Yaskawa INFORM job: OK_R2_O8A-O21A(90,0)OKKR.JBI

/JOB
//NAME OK_R2_O8A-O21A(90,0)OKKR
///FOLDERNAME X4
//POS
///NPOS 715,715,715,30,0,0
///TOOL 0
///POSTYPE PULSE
///PULSE
C00000=-132511,-103668,-126871,1472,79341,-68717
C00001=-132511,-105453,-125920,1479,77839,-68735
C00002=-149942,-121925,-119361,-5630,57848,-69572
C00003=-131289,-120708,-115141,-16553,58451,-62255
C00004=-130492,-107448,-108919,-16502,61476,-62404
C00005=-130492,-107531,-107691,-16624,60708,-62286
C00006=-130492,-107522,-107880,-16606,60824,-62304
C00007=-130122,-101219,-105586,-16530,62651,-62436
C00008=-130467,-107013,-108826,-16492,61638,-62417
C00009=-119884,-107962,-112031,-5369,66225,-56914
C00010=-116096,-92200,-106106,-6995,70935,-55838
C00011=-116096,-92633,-105187,-7026,70153,-55791
C00012=-116096,-92564,-105343,-7022,70283,-55799
C00013=-116785,-88340,-103625,-6657,71334,-56095
C00014=-116573,-89121,-105150,-6736,71883,-56054
C00015=-146016,-80865,-95606,32019,76533,-60687
C00016=-144125,-79506,-95002,31288,76137,-60071
C00017=-145805,-80719,-95541,31939,76487,-60619
C00018=-143803,-87593,-101078,23589,73333,-61663
C00019=-130467,-106338,-112373,-16140,64070,-62776
C00020=-173804,-84257,-100337,8034,65857,-78258
C00021=-173658,-84030,-99866,7982,65672,-78220
C00022=-173658,-84451,-98929,8028,64885,-78273
C00023=-173658,-84370,-99117,8019,65041,-78263
C00024=-172100,-80256,-97322,7106,65901,-77657
C00025=-174189,-84275,-102553,8181,67232,-78295
C00026=-146680,-106555,-114552,-7207,63010,-68642
C00027=-194694,-79170,-110255,-25784,98520,48468
C00028=-198558,-80793,-107909,-24687,95396,47836
C00029=-200090,-81195,-106872,-24266,94212,47563
C00030=-202263,-84154,-108139,-23691,92956,47080
C00031=-202263,-85492,-106716,-23644,91519,47366
C00032=-203864,-86202,-108997,-23266,92055,46716
C00033=-200090,-81195,-106872,-24266,94212,47563
C00034=-174358,-91389,-89628,-58384,85447,80654
C00035=-175228,-93280,-90391,-58296,84646,80691
C00036=-174358,-91389,-89628,-58384,85447,80654
C00037=-168427,-86826,-93699,-59246,91643,79819
C00038=-162839,-83719,-106729,-43881,81993,66911
C00039=-147123,-91237,-114479,-20257,52031,49855
C00040=-112908,-124838,-130477,-22240,82773,36203
C00041=-117493,-120147,-121828,-21064,78888,35282
C00042=-131517,-88028,-114974,-8271,96172,30135
C00043=-131517,-89283,-114090,-8245,94996,30214
C00044=-131517,-88930,-114352,-8253,95335,30191
C00045=-131178,-82908,-111873,-8367,96921,30191
C00046=-131517,-87249,-115462,-8285,96867,30089
C00047=-132831,-90163,-114266,-11578,93705,29175
C00048=-134095,-89636,-114054,-11263,93680,28777
C00049=-131312,-89742,-115220,-11972,94693,29560
C00050=-110699,-95947,-121920,-22827,92218,35184
C00051=-159423,-136044,-122705,-19473,51748,49954
C00052=-156084,-144100,-135379,-20578,56007,50549
C00053=-159635,-139405,-132559,-18260,112136,84879
C00054=-178843,-153016,-133090,-20490,101295,79475
C00055=-178843,-153131,-133279,-20494,101347,79466
C00056=-178843,-151887,-131264,-20445,100783,79562
C00057=-178843,-153131,-133279,-20494,101347,79466
C00058=-178681,-162456,-135669,-20227,98263,80057
C00059=-165549,-147119,-131679,-18745,106518,83551
C00060=-164263,-165353,-136391,-17937,100651,41944
C00061=-168242,-162829,-132237,-18538,98565,40818
C00062=-170474,-158220,-131092,-19006,99630,39839
C00063=-168242,-162829,-132237,-18538,98565,40818
C00064=-163940,-146805,-133599,-18623,108164,40895
C00065=-162398,-133850,-130940,-19068,113277,40626
C00066=-162571,-113567,-127717,-17378,114163,86924
C00067=-160654,-117481,-127396,-16916,112431,87902
C00068=-160654,-117651,-127195,-16888,112229,87933
C00069=-160654,-118532,-125995,-16733,111086,88103
C00070=-160654,-118346,-126273,-16766,111343,88065
C00071=-161650,-123459,-127890,-16641,109583,87959
C00072=-158594,-113131,-127392,-17075,114977,88272
C00073=-174543,-100010,-122844,-18621,115499,82286
C00074=-174543,-100010,-122844,-18621,115499,82286
C00075=-174543,-100010,-122844,-18621,115499,22315
C00076=-138816,-129701,-130055,-13678,112254,36070
C00077=-137500,-131474,-125884,-13183,109137,36932
C00078=-137500,-131471,-125777,-13177,109074,36939
C00079=-139149,-130411,-125460,-13458,109147,36324
C00080=-137500,-131471,-125777,-13177,109074,36939
C00081=-137500,-129047,-134180,-13875,115320,36192
C00082=-137500,-130207,-132407,-13667,113680,36396
C00083=-137899,-129904,-132317,-13740,113712,36243
C00084=-137899,-129904,-132317,-13740,113712,68510
C00085=-153549,-123160,-126704,-15778,110958,63049
C00086=-153549,-123239,-126516,-15760,110807,63070
C00087=-153549,-123761,-124983,-15622,109641,63231
C00088=-153549,-123239,-126516,-15760,110807,63070
C00089=-162223,-110280,-122283,-17095,113025,59536
C00090=-162223,-111585,-120346,-16843,111240,59807
C00091=-163386,-116637,-122034,-16744,109515,59637
C00092=-162108,-110157,-121578,-17034,112692,59632
C00093=-164629,-100924,-122013,-18009,116976,58006
C00094=-164629,-100924,-122013,-18009,116976,86315
C00095=-166469,-102657,-116169,-17620,113433,86211
C00096=-165427,-104649,-116407,-17406,112807,86697
C00097=-165427,-101226,-120322,-18070,116786,86050
C00098=-165427,-100996,-120510,-18111,117009,86012
C00099=-148525,-143011,-136643,3983,84771,-6637
C00100=-128066,-147732,-136598,30045,86114,-11272
C00101=-107762,-175532,-134890,18909,55578,3499
C00102=-107762,-174389,-134000,18900,55616,3506
C00103=-107762,-171707,-131824,18892,55653,3513
C00104=-107762,-174389,-134000,18900,55616,3506
C00105=-110240,-168768,-132692,19371,58166,2939
C00106=-107762,-174389,-134000,18900,55616,3506
C00107=-136558,-139033,-124155,30771,85335,-13620
C00108=-136645,-139245,-122439,30816,84359,-13917
C00109=-135016,-140023,-122655,30663,83532,-13499
C00110=-136645,-139245,-122439,30816,84359,-13917
C00111=-136645,-142239,-130726,30739,87441,-13088
C00112=-136645,-142239,-130726,30739,87441,-13088
C00113=-136231,-126717,-125654,30746,91494,-11840
C00114=-98133,-136848,-119853,-8087,80711,-399
C00115=-120576,-107226,-130969,4806,98429,26759
C00116=-134040,-103912,-127141,12417,95216,42526
C00117=-135128,-102736,-122709,12628,93295,41985
C00118=-135270,-98410,-119352,12667,93467,41957
C00119=-135270,-99211,-118697,12651,92671,41876
C00120=-135270,-98984,-118890,12655,92901,41899
C00121=-134962,-94751,-117294,12605,94023,42111
C00122=-135502,-100967,-121058,12716,93242,41857
C00123=-134459,-102900,-122675,12466,93098,42180
C00124=-132900,-95838,-124142,12211,97313,43092
C00125=-133104,-101231,-126476,12555,90730,41824
C00126=-142488,-103018,-116603,-18920,70477,-33231
C00127=-149408,-93922,-109008,-15541,69095,-35470
C00128=-149408,-94512,-107956,-15635,68178,-35347
C00129=-149408,-94372,-108222,-15611,68405,-35378
C00130=-148690,-90146,-106536,-15855,69631,-35290
C00131=-149408,-93897,-109054,-15536,69135,-35476
C00132=-123067,-90692,-110186,-27168,77789,-27787
C00133=-102416,-91941,-110630,-34518,86135,-22666
C00134=-101917,-92285,-106963,-34730,79171,-22421
C00135=-101917,-92861,-105821,-34832,78340,-22159
C00136=-102166,-91294,-105409,-34682,78702,-22372
C00137=-102552,-87773,-103968,-34461,79319,-22719
C00138=-102166,-90677,-106542,-34586,79544,-22637
C00139=-88745,-139673,-123014,-32701,61923,-22452
C00140=-91020,-118461,-119227,-25559,70043,-27274
C00141=-91020,-118666,-117531,-25735,69003,-27036
C00142=-91020,-118652,-117696,-25718,69101,-27059
C00143=-92656,-112693,-115717,-24791,70291,-27955
C00144=-91020,-118652,-117696,-25718,69101,-27059
C00145=-83494,-110253,-114881,-28187,73796,-25285
C00146=-83494,-110339,-114551,-28219,73576,-25230
C00147=-84308,-111339,-114895,-27963,73042,-25409
C00148=-86719,-114160,-115853,-27192,71497,-25959
C00149=-85916,-112867,-117155,-27291,73063,-26031
C00150=-123117,-127863,-126220,-28315,69551,-25784
C00151=-125315,-122167,-126738,-14196,74486,-31169
C00152=-125647,-109964,-126758,6698,85320,-36650
C00153=-127309,-126191,-121158,24496,77378,-41430
C00154=-122509,-120998,-116871,23174,76039,-39921
C00155=-117160,-104372,-112630,18566,82677,-37125
C00156=-117160,-104907,-110988,18612,81456,-37312
C00157=-117160,-104733,-111581,18595,81887,-37246
C00158=-112842,-111563,-113988,14481,77147,-33000
C00159=-113063,-106504,-112219,14479,78650,-32898
C00160=-112842,-111563,-113988,14481,77147,-33000
C00161=-122612,-110522,-114147,22924,79491,-39282
C00162=-127138,-114707,-118233,24171,81082,-40600
C00163=-112168,-135147,-125869,19703,71474,-13622
C00164=-107112,-124941,-122811,17686,73526,-11445
C00165=-98892,-86649,-110918,2998,94873,14107
C00166=-112057,-63273,-99647,16927,107898,-6848
C00167=-111820,-63961,-99109,16821,107199,-6872
C00168=-111820,-65039,-98309,16715,106195,-7017
C00169=-111820,-64914,-98405,16727,106313,-7000
C00170=-110559,-64565,-98232,16557,106153,-6607
C00171=-111820,-64402,-98791,16776,106793,-6930
C00172=-102401,-90236,-113117,-129,94163,18304
C00173=-122722,-94557,-112635,4536,92169,11873
C00174=-122722,-95060,-112012,4533,91529,11850
C00175=-122722,-94938,-112169,4534,91688,11856
C00176=-124421,-94788,-112110,4914,91823,11321
C00177=-122722,-94458,-112752,4538,92292,11877
C00178=-121995,-82445,-116286,4470,100580,12401
C00179=-106227,-105095,-124470,-409,77251,17488
C00180=-147196,-120547,-129970,-14917,75808,13222
C00181=-161004,-130220,-121828,-20444,67155,12825
C00182=-163784,-117907,-115753,-19016,68936,11464
C00183=-171500,-102190,-112609,-10247,77482,8342
C00184=-172766,-99537,-110960,-8908,78464,7982
C00185=-164799,-113448,-113379,-18515,69495,10996
C00186=-160173,-111708,-112729,-20272,71037,12446
C00187=-159937,-107532,-111273,-20230,72269,12319
C00188=-160173,-111708,-112729,-20272,71037,12446
C00189=-157530,-113449,-113320,-21331,71196,13397
C00190=-157502,-114878,-111335,-21583,69377,13748
C00191=-159463,-112600,-110567,-20755,69532,12980
C00192=-157502,-114878,-111335,-21583,69377,13748
C00193=-157530,-113449,-113320,-21331,71196,13397
C00194=-164799,-113448,-113379,-18515,69495,10996
C00195=-163784,-117907,-115753,-19016,68936,11464
C00196=-161004,-130220,-121828,-20444,67155,12825
C00197=-158635,-143974,-124952,-47178,64629,-48132
C00198=-161510,-136095,-119169,-46184,63472,-49060
C00199=-162608,-132555,-115350,-46042,62530,-49158
C00200=-162346,-131008,-113540,-46239,62439,-48970
C00201=-162608,-133192,-116899,-45817,62973,-49385
C00202=-136560,-74570,-80638,-73986,100743,-31924
C00203=-136560,-74368,-74379,-73183,99581,-30233
C00204=-138115,-75223,-74700,-73053,98436,-30293
C00205=-135508,-73752,-74143,-73275,100358,-30196
C00206=-149616,-145660,-96573,-81184,49972,-24507
C00207=-150329,-142641,-96001,-80244,49710,-25268
C00208=-148962,-149729,-97186,-82532,50127,-23453
C00209=-146770,-153464,-99018,-82858,51507,-22849
C00210=-140616,-162996,-103531,-83341,55379,-21287
C00211=-129649,-178931,-115518,-81569,62637,-20208
C00212=-149811,-117254,-127694,-14309,93218,-9052
C00213=-138773,-86779,-112433,-16512,101214,-6420
C00214=-139010,-84837,-109587,-16423,100448,-6393
C00215=-139010,-86284,-108173,-16326,98898,-6181
C00216=-139046,-85929,-108499,-16342,99259,-6242
C00217=-139851,-81484,-106752,-16280,100273,-6644
C00218=-139210,-85073,-109125,-16364,100022,-6400
C00219=-160229,-93267,-112119,-12359,94277,-12585
C00220=-159749,-92653,-111811,-12461,94470,-12448
C00221=-159749,-93339,-110977,-12438,93625,-12360
C00222=-159895,-92298,-111808,-12436,94626,-12511
C00223=-160151,-89339,-110624,-12406,95366,-12669
C00224=-159895,-92298,-111808,-12436,94626,-12511
C00225=-154010,-101242,-121994,-13665,97135,-10872
C00226=-154083,-100267,-121778,-13665,97483,-10934
C00227=-147006,-81102,-116195,-13282,100818,40144
C00228=-151269,-63896,-105225,-12354,102282,38687
C00229=-152138,-63686,-103764,-12097,101397,38514
C00230=-152138,-64898,-103136,-12048,100410,38612
C00231=-152138,-64707,-103240,-12056,100569,38597
C00232=-153752,-65312,-103536,-11647,100239,38140
C00233=-152274,-63472,-103683,-12067,101440,38470
C00234=-162010,-107602,-126737,-9369,91949,36281
C00235=-162010,-107602,-126737,-9369,91949,36281
C00236=-210314,-79584,-107375,35746,108623,-54127
C00237=-185587,-33049,-75742,32288,103518,-46434
C00238=-184078,-34029,-75535,31853,102480,-46201
C00239=-182552,-34930,-76118,31484,101891,-45830
C00240=-182816,-34825,-76051,31547,101988,-45895
C00241=-182831,-36048,-74896,31379,100842,-46225
C00242=-185721,-33305,-75942,32316,103553,-46472
C00243=-194611,-82272,-100926,32769,98332,-51304
C00244=-192673,-88198,-103442,32335,96357,-51142
C00245=-191529,-89685,-104055,32127,95614,-50921
C00246=-191825,-89362,-103923,32180,95794,-50983
C00247=-191825,-89971,-102555,32100,94805,-51265
C00248=-194745,-83421,-100673,32716,97748,-51530
C00249=-202657,-68845,-90344,38048,95727,-59775
C00250=-197239,-49375,-79846,37211,96371,-57406
C00251=-190625,-19292,-60428,35861,96684,-54792
C00252=-196048,-18383,-62081,37469,99924,-55713
C00253=-194745,-77273,-107470,33657,103946,-49656
C00254=-180005,-94840,-122299,-4648,94317,30566
C00255=-161456,-138612,-119355,-33475,60108,39853
C00256=-177811,-145909,-118581,-20235,46663,29920
C00257=-175917,-139954,-111417,-22701,46255,31618
C00258=-170439,-155606,-119968,-27049,45364,34664
C00259=-142804,-136998,-117626,-37100,63175,22857
C00260=-144648,-132967,-113782,-36586,62145,22385
C00261=-144885,-129361,-107588,-37135,60461,22914
C00262=-136947,-145476,-117578,-40176,62334,25990
C00263=-196282,-87995,-108739,-3579,85426,743
C00264=-205037,-102884,-106741,6782,68268,-1518
C00265=-216929,-66677,-95372,18946,93343,-19154
C00266=-227648,-50570,-80193,40663,106234,-15408
C00267=-214308,-78850,-94573,37906,96134,-13686
C00268=-212846,-79345,-94795,37666,95431,-13340
C00269=-188383,-103961,-111964,10748,79789,-11413
C00270=-188473,-109529,-112575,10859,77358,-11657
C00271=-187226,-109023,-106592,32700,78578,-8466
C00272=-176928,-85967,-103932,21600,91605,-23275
C00273=-179781,-73674,-98589,24940,98528,-27327
C00274=-188222,-67873,-108629,27686,109139,-27784
C00275=-193624,-62519,-106039,28903,111697,-28985
C00276=-181889,-64694,-107206,10450,102860,46697
C00277=-156132,-116840,-116416,-18883,68145,52042
C00278=-157304,-71640,-98542,-17370,79547,49887
C00279=-175414,-50228,-100699,8949,105606,48817
C00280=-160705,-81264,-118021,-1653,95624,51077
C00281=-127953,-81916,-111881,-42691,92562,-11616
C00282=-120615,-98718,-118071,-9470,89242,10072
C00283=-120614,-100809,-115874,-9471,86847,10254
C00284=-116758,-96041,-112477,-16669,91295,14808
C00285=-119673,-105427,-116369,-9746,84913,10709
C00286=-120613,-100772,-115937,-9471,86904,10250
C00287=-123745,-106180,-116020,-15024,87085,13022
C00288=-120614,-100813,-115850,-14161,89229,15792
C00289=-120615,-98722,-118044,-14185,91583,15523
C00290=-139593,-120017,-125917,-14274,80051,-13697
C00291=-147459,-122057,-122338,8250,71740,-26203
C00292=-147460,-122349,-119714,8332,69994,-26324
C00293=-146868,-122707,-118464,8148,68992,-26179
C00294=-147775,-127178,-120450,8566,68018,-26578
C00295=-149021,-123014,-119622,8969,69764,-26896
C00296=-147824,-122334,-115361,8622,67385,-26641
C00297=-147464,-122345,-117274,8412,68510,-26430
C00298=-147464,-122366,-119995,8326,70156,-26314
C00299=-147464,-118224,-129513,8030,78063,-25782
C00300=-147464,-118224,-129513,6689,118601,-78925
C00301=-147464,-118224,-129513,6689,118601,-90375
C00302=-129716,-111878,-123336,-3524,122371,-86039
C00303=-133010,-154239,-135553,-3817,108008,-86806
C00304=-90490,-99752,-122446,25205,102120,-77013
C00305=-92153,-96107,-120269,25526,103067,-77386
C00306=-91449,-165235,-132184,-12723,106899,-71864
C00307=-126355,-98414,-119449,-2829,127024,-84850
C00308=-140836,-122858,-129041,-139,116760,-83504
C00309=-161524,-153313,-130940,-22826,105718,-85992
C00310=-121833,-132425,-113961,44925,89262,-78761
C00311=-121169,-125555,-111250,44945,90266,-78000
C00312=-170754,-150027,-130781,-22970,104423,-89675
C00313=-173213,-138110,-133115,4817,110614,-73303
C00314=-177187,-122938,-126693,7576,117589,-76428
C00315=-178664,-97821,-112009,-32036,94837,-77481
C00316=-178457,-102445,-114055,-32005,93957,-77153
C00317=-182303,-120115,-123340,6380,117411,-78387
C00318=-196032,-116529,-119112,12805,118826,-82600
C00319=-182806,-113441,-126130,6638,122566,-78264
C00320=-165277,-120173,-132750,1498,117651,-75946
C00321=-206281,-102167,-121925,2944,121695,-77552
C00322=-201464,-114352,-117147,-5757,101650,67438
C00323=-200368,-109540,-114804,-5783,102752,67759
C00324=-201402,-116171,-127223,3466,115800,-80739
C00325=-193157,-133496,-132973,4059,108698,-85184
C00326=-168030,-129679,-131435,1038,111998,-77011
C00327=-152590,-129390,-129911,3156,110818,-71484
C00328=-141767,-123602,-126880,4599,111419,-67583
C00329=-141114,-115628,-126239,4831,115072,-67194
C00330=-147247,-120038,-130806,-8856,110749,-89640
C00331=-138147,-116215,-122144,-16955,111448,-87520
C00332=-136269,-107535,-118257,-19196,116051,-87125
C00333=-188488,-115235,-117264,8764,104512,67856
C00334=-187301,-109373,-114560,8881,105718,68358
C00335=-135583,-106226,-116474,-19024,115804,-86815
C00336=-137886,-102725,-119104,-19994,118513,-88211
C00337=-139135,-112852,-128624,-20291,118843,-88765
C00338=-139292,-114870,-129287,-20177,118215,-88704
C00339=-187982,-104318,-127456,3477,89797,72703
C00340=-187990,-108723,-124740,3481,85869,72593
C00341=-150971,-156992,-126089,-36978,57776,90090
C00342=-185963,-105163,-121881,2858,85864,73233
C00343=-188144,-110357,-123681,3535,84387,72501
C00344=-177479,-158791,-126402,-24830,46112,80956
C00345=-188029,-108820,-124772,3493,85841,72579
C00346=-188022,-104421,-127490,3489,89767,72690
C00347=-174298,-113219,-115861,-15770,66124,-24057
C00348=-180248,-105581,-114235,-5768,75934,-20428
C00349=-173939,-113739,-113379,-16158,64464,-23688
C00350=-174688,-117897,-113404,-16083,62276,-23658
C00351=-178039,-105217,-114293,-8002,76645,-18456
C00352=-176302,-111719,-108846,-15247,62325,-24289
C00353=-174039,-113317,-109052,-16445,62092,-23376
C00354=-172539,-113538,-108977,-17189,62243,-22815
C00355=-174267,-113511,-110133,-16253,62591,-23541
C00356=-174258,-113480,-112891,-16028,64241,-23777
C00357=-174307,-102252,-117157,-11533,81046,-15470
C00358=-174345,-102365,-117198,-11521,81009,-15479
C00359=-190775,-91857,-121708,11796,95177,-30723
C00360=-208754,-98864,-112717,37128,92966,-49075
C00361=-214846,-120327,-106837,51151,83157,-62011
C00362=-214841,-119670,-104864,51217,82591,-62323
C00363=-213748,-118658,-103835,51125,81907,-62125
C00364=-216770,-120620,-104459,51433,83201,-63007
C00365=-216373,-116987,-103296,51322,83714,-62508
C00366=-213511,-117312,-100524,51236,80910,-62555
C00367=-214845,-118750,-102310,51312,81889,-62717
C00368=-214851,-119483,-104312,51238,82440,-62412
C00369=-218178,-115538,-118233,49266,91982,-56948
C00370=-169784,-95533,-109053,46596,84452,16696
C00371=-175845,-105369,-102937,51834,73714,22623
C00372=-164097,-105161,-87202,73197,71611,28965
C00373=-156530,-108712,-88432,73008,66030,29334
C00374=-153715,-109814,-88807,72915,63973,29506
C00375=-170527,-92138,-98060,54392,80356,25101
C00376=-150294,-107027,-97281,61507,70646,37862
C00377=-161372,-116003,-107175,47183,64470,24730
C00378=-161496,-116499,-106623,47427,64124,24479
C00379=-160177,-94155,-100974,47088,76268,32721
C00380=-150157,-107158,-97564,61401,70593,37908
C00381=-149972,-107595,-97892,61293,70435,37894
C00382=-88166,-83507,-88464,28128,42437,57953
C00383=-81990,-163011,-124449,5585,29613,56921
C00384=-162881,-120047,-112782,46142,67476,23200
C00385=-153966,-116641,-122556,34655,76025,15464
C00386=-117008,-148876,-136987,-1466,73673,-38063
C00387=-126252,-131765,-130839,5463,89111,-40743
C00388=-164884,-144192,-115550,40419,81461,-56636
C00389=-155654,-112195,-105982,39074,85451,-51112
C00390=-119819,-85991,-113186,4537,101348,-38176
C00391=-122079,-96641,-122243,4925,101568,-38878
C00392=-101099,-87648,-113482,-27968,109543,44429
C00393=-96573,-127188,-118314,-27771,102918,48226
C00394=-85542,-184273,-129406,-35752,72010,61176
C00395=-93167,-147547,-121037,-33801,80320,55364
C00396=-110218,-114507,-123212,-16108,86718,46162
C00397=-152504,-138441,-132085,16664,78093,-9085
C00398=-191457,-109567,-125034,9426,80684,-19151
C00399=-214381,-113602,-114057,27955,63726,-64142
C00400=-214387,-113723,-111179,28386,62102,-64581
C00401=-214215,-113093,-109988,28405,61682,-64623
C00402=-214389,-113728,-111258,28375,62143,-64570
C00403=-212738,-111566,-109277,27620,61502,-64048
C00404=-213962,-113354,-110083,28305,61529,-64556
C00405=-213875,-114695,-110689,28343,61221,-64605
C00406=-214364,-113704,-111171,28374,62098,-64572
C00407=-214357,-113582,-114048,27943,63722,-64133
C00408=-174283,-101247,-119871,16121,93821,-65453
C00409=-173838,-102051,-118577,15993,92575,-65467
C00410=-173872,-98338,-116871,16021,93408,-65372
C00411=-175145,-99456,-118673,16315,94157,-65691
C00412=-174352,-103659,-116009,20693,93585,-64688
C00413=-174312,-103656,-117420,20719,94391,-64539
C00414=-176714,-116929,-126906,19302,86766,-16179
C00415=-181382,-121683,-127165,-5388,71552,-36447
C00416=-187446,-131805,-111566,-37879,40004,-62235
C00417=-187463,-129896,-107666,-38934,38872,-61621
C00418=-196931,-137408,-106251,-30039,25480,-61548
C00419=-186446,-131716,-107742,-40356,38644,-60793
C00420=-185573,-127298,-105247,-40377,39617,-60774
C00421=-195382,-135116,-104184,-30970,27320,-63567
C00422=-187457,-128566,-105102,-39647,38173,-61211
C00423=-187441,-130558,-109037,-38564,39279,-61835
C00424=-196640,-143323,-122728,-29866,37120,-66734
C00425=-185945,-125174,-129582,-39897,103153,-69319
C00426=-170870,-163570,-118040,-55029,81249,-52095
C00427=-212686,-113481,-89566,-12963,78888,71132
C00428=-215151,-115296,-90915,-12760,78396,70316
C00429=-179786,-150779,-115124,-54947,78878,-55682
C00430=-197696,-107272,-114471,-38964,97919,-72363
C00431=-152343,-113083,-118185,-24814,126675,-56048
C00432=-195513,-97078,-100361,-45515,122539,-78558
C00433=-215589,-109296,-82766,-10801,104809,70870
C00434=-212839,-110161,-82796,-9951,104741,71860
C00435=-197384,-92043,-95352,-45654,121244,-78899
C00436=-155394,-107237,-115802,-26414,127157,-57611
C00437=-147814,-144132,-130264,-24847,111600,-50742
C00438=-214385,-115050,-91121,-15616,71856,39505
C00439=-214401,-113114,-87216,-15735,70495,39681
C00440=-214407,-112311,-85637,-15785,69955,39751
C00441=-212607,-111613,-85852,-16057,70779,40304
C00442=-214366,-115000,-87352,-15823,69648,39808
C00443=-214392,-111585,-84244,-16055,65381,44584
C00444=-214410,-109897,-81022,-24415,69187,61260
C00445=-214414,-110066,-81336,-23540,70296,59097
C00446=-214409,-110914,-82947,-23467,70808,58993
C00447=-214399,-112969,-86931,-23295,72098,58733
C00448=-182860,-108511,-132060,-8820,106503,-33858
C00449=-240778,-137351,-128254,45983,85020,28938
C00450=-236675,-121649,-106302,61967,62621,57515
C00451=-232044,-114198,-104885,58168,72082,54237
C00452=-229664,-110741,-95811,60985,57497,58236
C00453=-229315,-118320,-101960,58791,68287,53156
C00454=-229655,-120240,-104287,58708,68736,53276
C00455=-234583,-97480,-91005,63317,70484,56777
C00456=-229776,-113988,-100474,59540,68570,54230
C00457=-228514,-118846,-102600,58604,67861,53364
C00458=-228397,-117924,-100288,58905,67278,52989
C00459=-228591,-117447,-99611,58998,67304,52880
C00460=-228007,-118154,-101138,58697,67254,53236
C00461=-227998,-119492,-104806,58168,68101,53893
C00462=-217117,-124631,-136943,31097,89965,17175
C00463=-212311,-124866,-133165,25299,83870,9309
C00464=-196995,-84615,-117906,-17381,99261,-54937
C00465=-196689,-87191,-114654,-17284,96138,-54393
C00466=-165175,-82845,-98210,-49348,99127,-47707
C00467=-196743,-87074,-114185,-17262,95909,-54377
C00468=-198014,-90395,-114090,-16887,93977,-54517
C00469=-178035,-61572,-88086,-47521,95827,-52133
C00470=-205373,-53531,-98850,-15247,101700,-58106
C00471=-205704,-49963,-101444,-15409,104963,-58624
C00472=-178318,-108601,-128727,-5603,100252,-45769
C00473=-168853,-122238,-134242,-1220,95726,-41713
C00474=-170297,-107383,-120290,24028,103073,-37740
C00475=-160733,-103929,-113030,25314,98004,-34995
C00476=-161047,-105719,-112436,25498,97896,-34186
C00477=-162344,-106453,-112811,25592,98148,-34602
C00478=-160733,-103887,-113137,25583,99045,-33815
C00479=-160980,-105216,-112985,19033,89759,-22187
C00480=-160982,-105144,-112901,20911,91577,-19207
C00481=-152566,-110009,-113460,-3309,75991,-4288
C00482=-157788,-107819,-112956,-241,74994,-7914
C00483=-120609,-111596,-118782,13024,86064,-14317
C00484=-133998,-113178,-111834,29794,79414,-36692
C00485=-133784,-113259,-111042,29784,78878,-36749
C00486=-133610,-109140,-109688,29638,79939,-36406
C00487=-135828,-112441,-110974,30250,79928,-37264
C00488=-134042,-113729,-112572,24695,80409,-36334
C00489=-133994,-113037,-113381,24636,81174,-36157
C00490=-133996,-112670,-115866,24554,82743,-35831
C00491=-134898,-132336,-126413,10595,74184,-11936
C00492=-133962,-121152,-121142,-2699,71953,10515
C00493=-133963,-121408,-118595,-2724,70256,10553
C00494=-134171,-122182,-117969,-2655,69467,10496
C00495=-132452,-124377,-118846,-3342,68943,11121
C00496=-134389,-126169,-119210,-2591,68176,10448
C00497=-130565,-111827,-114257,-5039,75994,15555
C00498=-126623,-133823,-126710,-6462,72649,17071
C00499=-133973,-119339,-126131,-2645,75950,10424
C00500=-158112,-98716,-126250,-19680,86530,-48527
C00501=-161036,-120263,-128161,-18992,76528,-47904
C00502=-158587,-105926,-119442,3034,92407,-44736
C00503=-161739,-127404,-118540,-19698,67291,-46630
C00504=-160544,-119732,-117016,-19776,70412,-46719
C00505=-162973,-178698,-129654,13234,43368,-49842
C00506=-139031,-178889,-128173,-23136,42482,-32605
C00507=-128071,-175110,-122136,-43612,45471,-24662
C00508=-147174,-158688,-112948,-50801,42531,-30258
C00509=-152757,-150397,-109355,-52122,42424,-31309
C00510=-171080,-122297,-124815,-15314,71519,-50716
C00511=-162896,-130847,-128779,-13430,60460,-45398
C00512=-130949,-94872,-120528,14594,85248,-55395
C00513=-53825,-116322,-125048,-14351,65953,-45020
C00514=30260,-81955,-85592,-10541,58194,89907
C00515=-126253,-78535,-68629,-1974,68777,60728
C00516=-133976,-48579,-51749,-422,66953,55442
C00517=-143445,-11852,-31053,1480,64717,48962
C00518=-147670,17027,-9476,9877,74622,49123
C00519=-147135,31900,7029,9795,72081,49101
C00520=-147059,31291,7516,9797,71470,49078
C00521=-147059,31341,6529,9765,72092,49129
C00522=-147727,26207,1471,9995,72641,48940
C00523=-147727,26139,2513,10029,71973,48885
C00524=-147511,27771,4102,9954,71808,48945
C00525=-147650,25585,2035,9999,71973,48912
C00526=-147650,26097,-2600,9851,75043,49164
C00527=-119782,42933,14409,5087,72220,53475
C00528=-118099,48860,22276,4468,70330,53985
C00529=-118099,48825,24454,4506,68976,53934
C00530=-118090,47987,23851,4504,68915,53935
C00531=-118090,48004,24664,4522,68425,53913
C00532=-118090,47958,23810,4504,68925,53935
C00533=-118049,44181,19766,4472,69469,53971
C00534=-118049,44151,20600,4487,68943,53949
C00535=-118075,46427,23028,4508,68620,53926
C00536=-118049,44122,20560,4487,68953,53949
C00537=-118049,44425,14984,4396,72529,54081
C00538=-116860,-24994,-46486,3887,74622,54555
C00539=-141580,-19095,-42244,13161,77572,46437
C00540=-154421,-19095,-42244,-7152,69599,54311
C00541=-168772,13045,-11724,-355,66689,49386
C00542=-168772,13045,-11724,-355,66689,49386
C00543=-178887,35491,12589,4659,63528,45673
C00544=-181596,22371,-6368,-6207,82852,43396
C00545=-180404,21966,-4986,-6100,81652,43706
C00546=-180404,21844,-4060,-6107,81025,43738
C00547=-180411,21948,-5012,-6098,81658,43703
C00548=-178663,19949,-6903,-6582,81925,44269
C00549=-178663,19811,-5890,-6592,81234,44305
C00550=-179639,22242,-3587,-6306,80996,43995
C00551=-178670,19793,-5916,-6590,81240,44302
C00552=-173498,18801,-6845,-8008,81758,45996
C00553=-173844,18831,-3651,-7950,79792,46005
C00554=-173838,18807,-2614,-7966,79149,46049
C00555=-173844,18768,-1984,-7975,78746,46073
C00556=-173844,18778,-2337,-7967,78964,46058
C00557=-174883,21039,-87,-7686,78645,45722
C00558=-173850,18758,-2365,-7965,78970,46055
C00559=-173850,19604,-9778,-7879,83922,45740
C00560=-173850,19604,-9778,-7879,54886,45740
C00561=-178844,-3710,-18963,-4726,48213,44074
C00562=-169145,-109680,-85477,-15638,36065,50412
C00563=-234460,-155557,-97015,52723,35880,9269
C00564=-234460,-155557,-97015,52723,35880,9269
C00565=-185005,-168424,-109045,51865,36378,9746
C00566=-146370,-47178,-55409,22603,47358,44094
C00567=-135046,22053,11,35916,47144,57269
C00568=-130494,57346,48467,50481,38778,58556
C00569=-131415,63711,60649,55587,36969,55624
C00570=-131415,64372,62385,56397,36549,55170
C00571=-131415,64150,61812,56128,36686,55320
C00572=-131562,59570,56520,55213,37300,55831
C00573=-131562,59864,57330,55590,37094,55619
C00574=-131480,62317,60156,56075,36770,55346
C00575=-131562,59864,57330,55590,37094,55619
C00576=-131448,57895,51970,52934,38342,56869
C00577=-110938,48639,31222,-8110,46478,55014
C00578=-110953,49007,15009,-7049,56559,54243
C00579=-121124,79167,29588,9119,86259,76275
C00580=-116364,78884,35462,-2572,70620,75042
C00581=-128168,96495,52619,20743,88473,62957
C00582=-128528,99904,58747,20832,86667,62522
C00583=-116510,76061,34871,-2667,67460,75035
C00584=-118808,65589,24299,-1737,65682,74224
C00585=-118576,74033,27538,-1707,72674,74215
C00586=-121440,87518,41247,10497,85367,68059
C00587=-105662,-52708,-103586,-702,92159,53545
C00588=-166025,-25947,-80013,26532,97101,31760
C00589=-164294,-17063,-34958,-31065,55273,-54461
C00590=-168124,42014,10128,-23159,81576,-60225
C00591=-168124,42014,10128,-23159,81576,-60225
C00592=-172939,75253,42203,-13683,94785,-62330
C00593=-173406,55787,34570,-11199,81413,-60765
C00594=-173520,53424,33189,-11186,81039,-60771
C00595=-171565,84309,54273,-17249,96185,-62349
C00596=-171160,78507,46357,-14030,96337,-61919
C00597=-169243,43363,4993,-17420,85083,-59919
C00598=-175926,65443,14304,-7549,79996,-66162
C00599=-175696,66112,18661,-7701,77698,-65949
C00600=-175037,96499,49818,-7828,90248,-66438
C00601=-175152,93287,46964,-7802,90342,-66481
C00602=-181384,57861,13137,4263,72611,-65787
C00603=-180472,61016,15404,5614,75426,-65150
C00604=-173823,64435,15621,-8474,78871,-65427
C00605=-163328,22111,-17695,-16319,60605,-55206
C00606=-158063,-10254,-35326,2776,53207,-35705
C00607=-177458,-62225,-50397,53512,41611,-19716
C00608=-177799,-66002,-78877,42886,52478,-23599
C00609=-139045,-15131,-45246,13545,58663,19299
C00610=-121149,62605,15567,-2560,83400,86983
C00611=-121104,37574,3044,-6249,65919,78986
C00612=-121857,39062,11359,-6061,61534,78949
C00613=-135865,87011,40718,24918,95497,56957
C00614=-136153,89985,46203,24876,93896,56517
C00615=-121170,40637,14511,-7670,60423,79126
C00616=-124590,33027,7905,-4581,58225,78083
C00617=-124019,34497,2441,-4724,64521,78018
C00618=-113341,59148,-2228,-3748,81595,52764
C00619=-104830,-47237,-107475,-6015,92389,46184
C00620=-168046,-22646,-92303,23676,100531,31319
C00621=-178506,-64043,-51330,54345,42002,-9320
C00622=-161820,24023,-17780,-7570,61243,-60628
C00623=-163544,81139,32356,-1868,89449,-65267
C00624=-166338,121298,87223,1460,91898,-67358
C00625=-158379,103529,59182,-8519,87603,-65182
C00626=-158357,100044,55900,-8524,87832,-65191
C00627=-165483,133833,104493,3316,90235,-66989
C00628=-165483,132536,100441,3322,92059,-66942
C00629=-165483,132698,96383,3323,92004,-66943
C00630=-164280,62524,18315,3678,70871,-65511
C00631=-164280,62524,18315,3678,70871,-65511
C00632=-167598,53802,18275,9750,60095,-66581
C00633=-143537,101175,57606,-16851,87230,-68252
C00634=-143394,97839,54544,-16884,87421,-68231
C00635=-164948,55848,19205,7089,61928,-65627
C00636=-164280,62524,18315,3678,70871,-65511
C00637=-158520,39777,460,-10756,55186,-64462
C00638=-156529,-359,-32075,2996,54939,-55409
C00639=-181545,-68424,-52291,57183,42847,-45278
C00640=-167548,-84726,-87643,38554,44554,-4966
C00641=-149856,11622,-36808,29194,79273,34001
C00642=-140029,48396,12731,1352,59561,70300
C00643=-140967,52440,26076,2383,52339,69844
C00644=-140151,91077,43318,-5378,90823,76333
C00645=-140389,94148,48975,-5317,88913,76337
C00646=-144356,48534,22725,5101,51530,68433
C00647=-142635,45115,7499,2961,61160,69375
C00648=-133313,28699,-18653,-10194,71920,51962
C00649=-133779,63712,17960,-31297,73149,1805
C00650=-186219,94953,45513,-14342,87588,-71362
C00651=-186395,93658,48045,-14309,85401,-71166
C00652=-180270,109525,69749,-22776,94906,-71476
C00653=-186672,90586,45814,-14233,85155,-71230
C00654=-186465,93628,48420,-14293,85151,-71161
C00655=-181283,116002,78799,-23871,93564,-71706
C00656=-181042,85607,34487,-24091,91898,-71547
C00657=-187973,97649,48980,-13845,86576,-71819
C00658=-178015,25801,-2762,-17551,60288,-59809
C00659=-181007,24336,5295,-13100,49316,-58766
C00660=-173162,91192,47015,-26597,96822,-52438
C00661=-173064,94370,49802,-26605,96778,-52392
C00662=-183228,26310,7248,-11564,48896,-59712
C00663=-180426,28912,2129,-16364,58448,-60464
C00664=-171125,56319,10086,-13223,80051,-64352
C00665=-165056,82559,28692,-10044,90073,-67966
C00666=-170548,119071,78932,2044,93213,-68624
C00667=-162801,94753,47772,-7506,90872,-66819
C00668=-162783,98187,53928,-7502,88866,-66693
C00669=-169631,117929,77290,1949,93613,-68313
C00670=-169847,118878,76938,1974,94323,-68374
C00671=-165711,116090,74970,1537,94015,-67008
C00672=-164478,115503,74186,1409,94174,-66599
C00673=-164732,116698,71039,1447,96730,-66653
C00674=-161581,95612,48921,-9384,78255,-63326
C00675=-163478,84936,35629,-5803,75686,-63247
C00676=-163283,74755,34461,-5395,65063,-62774
C00677=-161324,95565,53507,-9580,75474,-63025
C00678=-161323,99500,60299,-9673,73346,-62856
C00679=-166324,76155,36293,7696,65696,-62476
C00680=-166797,80537,31190,5547,74628,-62537
C00681=-176200,98212,51407,-7801,91214,-66899
C00682=-171637,111790,71602,-20426,99240,-67843
C00683=-176199,96277,49539,-7802,91368,-66909
C00684=-176031,99724,55728,-7827,89365,-66729
C00685=-168479,104724,61882,-19387,100817,-66832
C00686=-170338,96328,45386,-15093,101286,-66904
C00687=-175541,68734,11358,228,80553,-65403
C00688=-171596,79837,29569,-10570,74939,-65528
C00689=-175715,65983,24554,-1319,65350,-64997
C00690=-176205,96252,49495,-7801,91382,-66911
C00691=-176037,99696,55680,-7826,89379,-66732
C00692=-176721,74046,31552,7495,70864,-64311
C00693=-175645,84236,32364,2706,80895,-64352
C00694=-172106,73847,22038,-5154,77410,-64580
C00695=-171178,75490,24026,-5584,77087,-64273
C00696=-165276,24993,-49970,-8200,96948,-63695
C00697=-92014,-65792,-98654,-33564,68903,-44780
C00698=-92014,-65792,-98652,-33579,68908,-44779
C00699=-112544,25072,-21983,-21189,62436,-50668
C00700=-133924,64642,16887,-41400,76255,-73236
C00701=-139901,71761,28474,-30769,75742,-73566
C00702=-138936,75123,35778,-31507,73696,-72623
C00703=-141064,73190,33638,-30622,73223,-73319
C00704=-142367,96104,62019,-31075,67835,-72315
C00705=-144319,102422,66207,-23257,70324,-72918
C00706=-144704,106260,69701,-20057,71211,-72893
C00707=-142867,98447,59319,-20505,73887,-72688
C00708=-136902,87117,52885,-36282,86378,-76622
C00709=-135620,73631,40187,-40197,80568,-74982
C00710=-136624,86900,56391,-40286,77671,-74301
C00711=-134674,77415,38418,-40217,83337,-75634
C00712=-126958,42470,-7112,-42423,94399,-76801
C00713=-124399,-38669,-81065,-43564,98333,-77427
C00714=-15465,-107351,-121619,-48207,78518,-35388
BC00000=166351,717693,1075101
BC00001=124713,836357,1075101
BC00002=68993,906552,1075175
BC00003=68993,906552,1075175
BC00004=68993,906552,1075175
BC00005=68993,906552,1075175
BC00006=68993,906552,1075175
BC00007=68993,906552,1075175
BC00008=68993,906552,1075175
BC00009=68993,906552,1075175
BC00010=68993,906552,1075175
BC00011=68993,906552,1075175
BC00012=68993,906552,1075175
BC00013=68993,906552,1075175
BC00014=68993,906552,1075175
BC00015=68993,906552,1075175
BC00016=68993,906552,1075175
BC00017=68993,906552,1075175
BC00018=68993,906552,1075175
BC00019=68993,906552,1075175
BC00020=68993,906552,1075175
BC00021=68994,906552,1075171
BC00022=68994,906552,1075171
BC00023=68994,906552,1075171
BC00024=68994,906552,1075171
BC00025=68994,906552,1075171
BC00026=68993,906552,1075175
BC00027=168967,880191,1075175
BC00028=168967,880191,1075175
BC00029=168967,880191,1075175
BC00030=168967,880191,1075175
BC00031=168967,880191,1075175
BC00032=168967,880191,1075175
BC00033=168967,880191,1075175
BC00034=168967,880191,1075175
BC00035=168967,880191,1075175
BC00036=168967,880191,1075175
BC00037=168967,880191,1075175
BC00038=173610,886233,1075175
BC00039=182518,897827,1075175
BC00040=137300,943049,1075175
BC00041=137300,943049,1075175
BC00042=137300,943049,1075175
BC00043=137300,943049,1075175
BC00044=137300,943049,1075175
BC00045=137300,943049,1075175
BC00046=137300,943049,1075175
BC00047=137300,943049,1075175
BC00048=137300,943049,1075175
BC00049=137300,943049,1075175
BC00050=137300,943049,1075175
BC00051=206514,959231,1075175
BC00052=206514,959231,1075175
BC00053=192568,1039911,1075175
BC00054=191010,1035303,1075175
BC00055=191010,1035303,1075175
BC00056=191010,1035303,1075175
BC00057=191010,1035303,1075175
BC00058=191010,1035303,1075175
BC00059=191010,1035303,1075175
BC00060=199408,1035303,1075175
BC00061=199408,1035303,1075175
BC00062=199408,1035303,1075175
BC00063=199408,1035303,1075175
BC00064=199408,1035303,1075175
BC00065=249680,1035303,1075172
BC00066=249681,1035303,1075169
BC00067=249681,1035303,1075169
BC00068=249681,1035303,1075169
BC00069=249681,1035303,1075169
BC00070=249681,1035303,1075169
BC00071=249681,1035303,1075169
BC00072=249681,1035303,1075169
BC00073=249681,1035303,1075169
BC00074=249681,1035303,1075169
BC00075=249681,1035303,1075169
BC00076=249681,1035303,1075169
BC00077=249681,1035303,1075169
BC00078=249681,1035303,1075169
BC00079=249681,1035303,1075169
BC00080=249681,1035303,1075169
BC00081=249681,1035303,1075218
BC00082=249453,861783,1075169
BC00083=249453,861783,1075169
BC00084=249453,861783,1075169
BC00085=249453,861783,1075169
BC00086=249453,861783,1075169
BC00087=249453,861783,1075169
BC00088=249453,861783,1075169
BC00089=249453,861783,1075169
BC00090=249453,861783,1075169
BC00091=249453,861783,1075169
BC00092=249453,861783,1075169
BC00093=249453,861783,1075169
BC00094=249453,861783,1075169
BC00095=249453,861783,1075166
BC00096=249453,861783,1075166
BC00097=249453,861783,1075166
BC00098=249453,861783,1075198
BC00099=167652,857396,1075196
BC00100=42938,871634,1073896
BC00101=42938,871634,1073896
BC00102=42938,871634,1073896
BC00103=42938,871634,1073896
BC00104=42938,871634,1073896
BC00105=42938,871634,1073896
BC00106=42938,871634,1073896
BC00107=42938,871634,1073896
BC00108=42938,871634,1073896
BC00109=42938,871634,1073896
BC00110=42938,871634,1073896
BC00111=42938,871634,1073896
BC00112=211024,871590,1073896
BC00113=211024,871590,1073896
BC00114=216853,878500,1074004
BC00115=207524,931262,1074736
BC00116=201927,962915,1075175
BC00117=201927,962915,1075175
BC00118=201927,962915,1075175
BC00119=201927,962915,1075175
BC00120=201927,962915,1075175
BC00121=201927,962915,1075175
BC00122=201927,962915,1075175
BC00123=201927,962915,1075175
BC00124=201927,962915,1075175
BC00125=203493,945347,1075175
BC00126=350667,957415,1075175
BC00127=350667,957415,1075173
BC00128=350667,957415,1075173
BC00129=350667,957415,1075173
BC00130=350667,957415,1075173
BC00131=350667,957415,1075173
BC00132=350667,957415,1075175
BC00133=350667,957415,1075175
BC00134=350667,957415,1075175
BC00135=350667,957415,1075175
BC00136=350667,957415,1075175
BC00137=350667,957415,1075175
BC00138=350667,957415,1075175
BC00139=398035,984166,1075175
BC00140=398035,984166,1075175
BC00141=398035,984166,1075175
BC00142=398035,984166,1075175
BC00143=398035,984166,1075174
BC00144=398035,984166,1075175
BC00145=398035,984166,1075175
BC00146=398035,984166,1075175
BC00147=398035,984166,1075175
BC00148=398035,984166,1075175
BC00149=398035,984166,1075175
BC00150=350667,957415,1075175
BC00151=334076,958261,1075175
BC00152=306358,959675,1075175
BC00153=283206,960856,1075175
BC00154=283206,960856,1075175
BC00155=283206,960856,1075175
BC00156=283206,960856,1075175
BC00157=283206,960856,1075175
BC00158=283206,960856,1075175
BC00159=283206,960856,1075175
BC00160=283206,960856,1075175
BC00161=283206,960856,1075175
BC00162=283206,960856,1075175
BC00163=292069,950355,1075175
BC00164=292069,950355,1075175
BC00165=338620,875919,1075175
BC00166=338620,875919,1075175
BC00167=338620,875919,1075175
BC00168=338620,875919,1075175
BC00169=338620,875919,1075175
BC00170=338620,875919,1075175
BC00171=338620,875919,1075175
BC00172=338620,875919,1075175
BC00173=338620,875919,1075175
BC00174=338620,875919,1075175
BC00175=338620,875919,1075175
BC00176=338620,875919,1075175
BC00177=338620,875919,1075175
BC00178=338620,875919,1075175
BC00179=304928,940692,1075175
BC00180=308914,936786,1075174
BC00181=310258,935470,1075175
BC00182=310258,935470,1075175
BC00183=310258,935470,1075175
BC00184=310258,935470,1075175
BC00185=310258,935470,1075175
BC00186=310258,935470,1075175
BC00187=310258,935470,1075175
BC00188=310258,935470,1075175
BC00189=310258,935470,1075175
BC00190=310258,935470,1075175
BC00191=310258,935470,1075175
BC00192=310258,935470,1075175
BC00193=310258,935470,1075175
BC00194=310258,935470,1075175
BC00195=310258,935470,1075175
BC00196=310258,935470,1075175
BC00197=123812,849710,1075175
BC00198=123812,849710,1075175
BC00199=123812,849710,1075175
BC00200=123812,849710,1075175
BC00201=123812,849710,1075175
BC00202=123812,849710,1075175
BC00203=123812,849710,1075175
BC00204=123812,849710,1075175
BC00205=123812,849710,1075175
BC00206=123812,849710,1075175
BC00207=123812,849710,1075175
BC00208=123812,849710,1075175
BC00209=123812,849710,1075175
BC00210=123812,849710,1075175
BC00211=123812,849710,1075175
BC00212=123812,849710,1075175
BC00213=123812,849710,1075175
BC00214=123812,849710,1075175
BC00215=123812,849710,1075175
BC00216=123812,849710,1075175
BC00217=123812,849710,1075175
BC00218=123812,849710,1075175
BC00219=123812,849710,1075175
BC00220=123812,849710,1075175
BC00221=123812,849710,1075175
BC00222=123812,849710,1075175
BC00223=123812,849710,1075175
BC00224=123812,849710,1075175
BC00225=123812,849710,1075175
BC00226=123812,849710,1075175
BC00227=123812,849710,1075175
BC00228=123812,849710,1075175
BC00229=123812,849710,1075175
BC00230=123812,849710,1075175
BC00231=123812,849710,1075175
BC00232=123812,849710,1075175
BC00233=123812,849710,1075175
BC00234=123812,849710,1075175
BC00235=39173,787424,1075175
BC00236=39173,787424,1075175
BC00237=39173,787424,1075175
BC00238=39173,787424,1075175
BC00239=39173,787424,1075175
BC00240=39173,787424,1075175
BC00241=39173,787424,1075175
BC00242=39173,787424,1075175
BC00243=39173,787424,1075175
BC00244=39173,787424,1075175
BC00245=39173,787424,1075175
BC00246=39173,787424,1075175
BC00247=39173,787424,1075175
BC00248=39173,787424,1075175
BC00249=66331,782733,1075175
BC00250=66331,782733,1075175
BC00251=66331,782733,1075175
BC00252=66331,782733,1075175
BC00253=39173,787424,1075175
BC00254=123812,849710,1075175
BC00255=123812,849710,1075175
BC00256=123812,849710,1075175
BC00257=123812,849710,1075171
BC00258=123812,849710,1075171
BC00259=141948,851290,1075172
BC00260=141948,851290,1075172
BC00261=141948,851290,1075172
BC00262=141948,851290,1075172
BC00263=141948,851290,1075172
BC00264=141948,851290,1075172
BC00265=141948,851290,1075172
BC00266=141948,851290,1075172
BC00267=141948,851290,1075172
BC00268=141948,851290,1075172
BC00269=141948,851290,1075172
BC00270=141948,851290,1075172
BC00271=141948,851290,1075172
BC00272=141948,851290,1075172
BC00273=141948,851290,1075172
BC00274=141948,851290,1075172
BC00275=141948,851290,1075172
BC00276=141948,851290,1075172
BC00277=141949,851290,1075171
BC00278=141949,851290,1075171
BC00279=141948,851290,1075172
BC00280=141948,851290,1075172
BC00281=176393,854291,1075175
BC00282=222055,900780,1075175
BC00283=219754,905761,1075175
BC00284=226754,912438,1075175
BC00285=218833,907753,1075175
BC00286=218833,907753,1075175
BC00287=226754,912438,1075175
BC00288=221540,906670,1075175
BC00289=224964,902325,1075175
BC00290=248834,904813,1075175
BC00291=216311,894179,1075175
BC00292=217838,899796,1075175
BC00293=218449,902042,1075174
BC00294=218449,902043,1075175
BC00295=218449,902043,1075175
BC00296=215173,900211,1075175
BC00297=214562,897964,1075175
BC00298=213035,892347,1075175
BC00299=213035,892347,1075175
BC00300=213035,892347,1075175
BC00301=213035,1030309,1075175
BC00302=213035,1030309,1075175
BC00303=213035,1045492,1075175
BC00304=114747,944581,1036622
BC00305=114747,944581,1036622
BC00306=213035,1057569,1075175
BC00307=213035,1030309,1075175
BC00308=213035,1030309,1075175
BC00309=253909,1070223,1075174
BC00310=108163,941106,1075175
BC00311=108163,941106,1075175
BC00312=250408,1066805,1075174
BC00313=213035,1030309,1075175
BC00314=213035,1030309,1075175
BC00315=317025,983389,1075175
BC00316=317025,983389,1075175
BC00317=213035,1030309,1075175
BC00318=213035,1030309,1075175
BC00319=213035,1030309,1075175
BC00320=139079,982225,1075175
BC00321=139079,982225,1072947
BC00322=214992,960257,1075175
BC00323=214992,960257,1075175
BC00324=139079,982225,1072947
BC00325=139079,982225,1072947
BC00326=139079,982225,1072947
BC00327=139079,982225,1072947
BC00328=139079,982225,1072947
BC00329=139079,982225,1072947
BC00330=179211,989169,1072947
BC00331=179211,989169,1074170
BC00332=179211,989169,1074170
BC00333=161178,915980,1075175
BC00334=161178,915980,1075175
BC00335=179211,989169,1074170
BC00336=179211,989169,1074170
BC00337=179211,995679,1074170
BC00338=246769,865802,1074170
BC00339=94949,849781,1075175
BC00340=94241,849617,1075175
BC00341=93963,849554,1075173
BC00342=93964,849553,1075175
BC00343=93964,849553,1075175
BC00344=93963,849554,1075173
BC00345=74766,838694,1075175
BC00346=75473,838858,1075175
BC00347=233067,883965,1075175
BC00348=197070,880962,1075175
BC00349=228487,890641,1075175
BC00350=228487,890641,1075175
BC00351=220268,893974,1075175
BC00352=254174,905057,1075175
BC00353=254174,905057,1075173
BC00354=254174,905057,1075173
BC00355=255482,903149,1075175
BC00356=258754,898381,1075175
BC00357=225061,887890,1075175
BC00358=201863,874878,1075175
BC00359=178980,869980,1075175
BC00360=153940,864621,1075175
BC00361=139418,861513,1075175
BC00362=143006,867556,1075175
BC00363=144440,869973,1075175
BC00364=144440,869973,1075175
BC00365=144440,869973,1075175
BC00366=144438,869977,1075175
BC00367=143003,867560,1075175
BC00368=139416,861518,1075175
BC00369=144128,864459,1075175
BC00370=253458,932694,1075175
BC00371=273251,945047,1075175
BC00372=228147,945047,1075175
BC00373=228147,945047,1075175
BC00374=228147,945047,1075175
BC00375=273251,945047,1075175
BC00376=225208,952218,1075175
BC00377=273917,948573,1075175
BC00378=273917,948573,1075175
BC00379=273653,947175,1075175
BC00380=257870,958024,1075196
BC00381=310163,967320,1075229
BC00382=310203,967362,1075229
BC00383=345475,1000313,1075174
BC00384=365822,963946,1075175
BC00385=376741,960844,1075175
BC00386=370656,944994,1075175
BC00387=370656,892039,1075175
BC00388=370656,895716,1075174
BC00389=370656,895716,1075174
BC00390=370656,892039,1075175
BC00391=370656,892039,1075175
BC00392=370656,892039,1075175
BC00393=370656,921345,1075175
BC00394=370656,921345,1075175
BC00395=370656,921345,1075175
BC00396=370656,892039,1075175
BC00397=386422,918220,1075175
BC00398=361265,958626,1075175
BC00399=315393,987553,1075175
BC00400=315079,993002,1075175
BC00401=314955,995155,1075175
BC00402=314954,995181,1075175
BC00403=314954,995181,1075175
BC00404=319656,995999,1075175
BC00405=323151,996606,1075175
BC00406=324672,994669,1075175
BC00407=324985,989220,1075175
BC00408=237585,981036,1075175
BC00409=238823,981788,1075175
BC00410=238823,981788,1075175
BC00411=238823,981788,1075175
BC00412=223382,978120,1075175
BC00413=221852,977368,1075175
BC00414=241515,960881,1075175
BC00415=320615,986057,1075175
BC00416=360079,1022519,1075175
BC00417=355351,1023517,1075175
BC00418=353460,1023916,1075175
BC00419=353460,1023916,1075175
BC00420=353460,1023916,1075175
BC00421=357559,1021820,1075175
BC00422=359451,1021421,1075175
BC00423=364179,1020424,1075175
BC00424=364179,1020424,1075175
BC00425=304607,908316,1075175
BC00426=304607,908316,1075175
BC00427=288616,851871,1075175
BC00428=288616,851871,1075175
BC00429=304607,908316,1075175
BC00430=304607,908316,1075175
BC00431=231979,880249,1075172
BC00432=262921,926617,1075172
BC00433=233663,865189,1075175
BC00434=233663,865189,1075175
BC00435=262921,926617,1075172
BC00436=231979,880249,1075172
BC00437=231979,880249,1075172
BC00438=326594,857424,1075229
BC00439=323136,853802,1075229
BC00440=321752,852354,1075229
BC00441=321752,852354,1075229
BC00442=321752,852354,1075229
BC00443=328084,850016,1075229
BC00444=323279,867664,1075229
BC00445=321786,867486,1075229
BC00446=322406,869351,1075229
BC00447=323957,874014,1075229
BC00448=233836,901031,1075172
BC00449=238710,955570,1075175
BC00450=239384,978190,1075175
BC00451=219723,976819,1075175
BC00452=222174,977409,1075175
BC00453=219425,978744,1075175
BC00454=219425,978744,1075175
BC00455=222174,977409,1075175
BC00456=223674,978551,1075175
BC00457=224097,978873,1075175
BC00458=242049,979368,1075175
BC00459=246721,979497,1075175
BC00460=247019,977572,1075175
BC00461=247764,972760,1075175
BC00462=209134,929318,1075175
BC00463=202136,921448,1075175
BC00464=139989,851558,1075175
BC00465=139989,851558,1075175
BC00466=139989,851558,1075175
BC00467=139989,851558,1075175
BC00468=139989,851558,1075175
BC00469=139989,851558,1075175
BC00470=139989,851558,1075175
BC00471=139989,851558,1075175
BC00472=212582,902134,1075175
BC00473=254744,926256,1075175
BC00474=341543,975915,1075175
BC00475=346125,974361,1075175
BC00476=346334,977329,1075175
BC00477=346334,977329,1075175
BC00478=346334,977329,1075175
BC00479=364185,966891,1075175
BC00480=354904,971109,1075175
BC00481=391862,967110,1075171
BC00482=398174,963874,1075175
BC00483=310323,960378,1075175
BC00484=300015,957089,1075175
BC00485=301970,958289,1075175
BC00486=302239,958454,1075175
BC00487=302239,958454,1075175
BC00488=309604,960702,1075175
BC00489=307558,959354,1075175
BC00490=302443,955986,1075175
BC00491=333839,953225,1075175
BC00492=361939,950754,1075175
BC00493=359473,956199,1075175
BC00494=358656,958004,1075175
BC00495=358487,958377,1075175
BC00496=358487,958377,1075175
BC00497=358656,958004,1075175
BC00498=358656,958004,1075175
BC00499=361939,905440,1073950
BC00500=121221,890837,1075175
BC00501=121221,957471,1075175
BC00502=121221,957471,1075175
BC00503=120731,958579,1075175
BC00504=120731,958579,1075175
BC00505=121221,957471,1075175
BC00506=121221,957471,1075175
BC00507=121221,957471,1075175
BC00508=120732,958578,1075172
BC00509=65841,949070,1075175
BC00510=65841,949070,1075175
BC00511=66331,923914,1075175
BC00512=148919,744039,1075175
BC00513=196589,721705,1075175
BC00514=204899,695380,820586
BC00515=194375,692487,359056
BC00516=192469,726487,275453
BC00517=190132,768172,172952
BC00518=190132,768172,172952
BC00519=190132,768172,172952
BC00520=190132,768172,172952
BC00521=190132,768172,172952
BC00522=190132,768172,172952
BC00523=190132,768172,172952
BC00524=190132,768172,172952
BC00525=190132,768172,172952
BC00526=190132,768172,172952
BC00527=151334,768172,172952
BC00528=151334,768172,172952
BC00529=151334,768172,172952
BC00530=151334,768172,172952
BC00531=151334,768172,172952
BC00532=151334,768172,172952
BC00533=151334,768172,172952
BC00534=151334,768172,172952
BC00535=151334,768172,172952
BC00536=151334,768172,172952
BC00537=151334,768172,172952
BC00538=151334,768172,172952
BC00539=195455,768172,172952
BC00540=195455,768172,172952
BC00541=227925,768172,172952
BC00542=217420,785287,172952
BC00543=217420,804358,172952
BC00544=217420,804358,172952
BC00545=218636,803490,170876
BC00546=218636,803490,170876
BC00547=218636,803490,170876
BC00548=218636,803490,170876
BC00549=218636,803490,170876
BC00550=218636,803490,170872
BC00551=218636,803490,170876
BC00552=218636,803490,170876
BC00553=218636,803490,170876
BC00554=218636,803490,170876
BC00555=218636,803490,170876
BC00556=218636,803490,170876
BC00557=218636,803490,170876
BC00558=218636,803490,170876
BC00559=218636,803490,170876
BC00560=218636,803490,170876
BC00561=218636,803490,170876
BC00562=218636,803490,170876
BC00563=218636,803490,170876
BC00564=368953,803490,170876
BC00565=368953,803490,170876
BC00566=346770,805721,162531
BC00567=318847,808530,152027
BC00568=304865,809937,146768
BC00569=304865,809937,146767
BC00570=304865,809937,146767
BC00571=304865,809937,146767
BC00572=304865,809937,146767
BC00573=304865,809937,146767
BC00574=304865,809937,146767
BC00575=304865,809937,146767
BC00576=304773,809946,146732
BC00577=292507,811180,142119
BC00578=292507,811180,142119
BC00579=301416,829352,4514
BC00580=301416,815080,4514
BC00581=302510,828599,53
BC00582=302510,828599,53
BC00583=301416,815054,4514
BC00584=301416,814793,4514
BC00585=301416,814750,4514
BC00586=302510,816592,53767
BC00587=257688,677496,16011
BC00588=249672,677703,34632
BC00589=237199,771258,142432
BC00590=237199,771258,142432
BC00591=237199,771258,142432
BC00592=237199,771258,120395
BC00593=237200,771259,219475
BC00594=237200,771259,219475
BC00595=237199,771258,120395
BC00596=237199,771258,120395
BC00597=237199,771258,120395
BC00598=251479,761965,53
BC00599=251479,761965,53
BC00600=251479,761965,53
BC00601=251479,761965,53
BC00602=251479,761965,53
BC00603=251479,761965,53
BC00604=251479,761965,53
BC00605=241857,743783,27173
BC00606=220919,704221,86183
BC00607=190132,678003,172952
BC00608=333043,678806,172952
BC00609=321753,695280,153695
BC00610=297117,802708,111674
BC00611=285421,819898,121816
BC00612=285421,819898,121816
BC00613=284385,821419,53
BC00614=284385,821419,53
BC00615=285421,819898,121816
BC00616=285421,819898,121816
BC00617=285421,819898,121816
BC00618=260189,684435,56004
BC00619=252442,679825,35798
BC00620=252442,683048,35798
BC00621=190132,680512,172952
BC00622=239488,732658,34145
BC00623=239488,732658,34145
BC00624=239488,732658,34145
BC00625=251613,723934,53
BC00626=251613,723934,53
BC00627=239488,732658,34145
BC00628=239488,732658,34145
BC00629=239488,732658,34145
BC00630=232113,730739,27801
BC00631=232113,730739,27801
BC00632=232113,730739,27801
BC00633=199854,722343,53
BC00634=199854,722343,53
BC00635=232113,730739,27801
BC00636=232113,730739,27801
BC00637=232113,730739,27801
BC00638=219889,706079,70066
BC00639=190132,687376,172952
BC00640=333043,680581,172952
BC00641=325640,711150,89779
BC00642=315806,785654,86936
BC00643=315806,785654,86936
BC00644=313707,801555,53
BC00645=313707,801555,53
BC00646=315806,785654,86936
BC00647=315806,785654,86936
BC00648=316651,770280,62653
BC00649=318784,731458,1334
BC00650=382011,827237,53
BC00651=382011,827237,53
BC00652=360424,827237,53
BC00653=382011,827237,53
BC00654=382011,827237,53
BC00655=360424,827237,53
BC00656=360424,827237,53
BC00657=382011,827237,53
BC00658=335002,829407,125095
BC00659=335002,829407,125095
BC00660=335002,829687,53
BC00661=335002,829687,53
BC00662=335002,829407,125095
BC00663=335002,829407,125095
BC00664=349089,814359,67200
BC00665=365426,796907,50
BC00666=365426,796907,50
BC00667=365426,796907,53
BC00668=365426,796907,53
BC00669=365426,796907,50
BC00670=365426,796907,50
BC00671=365426,796907,50
BC00672=365426,796907,50
BC00673=365426,796907,50
BC00674=365650,790459,53
BC00675=365650,790459,53
BC00676=365650,790459,53
BC00677=365650,790459,53
BC00678=365650,790459,53
BC00679=365650,790459,53
BC00680=365650,790459,53
BC00681=367722,807347,53
BC00682=358204,818181,53
BC00683=367722,807347,53
BC00684=367722,807347,53
BC00685=358204,818181,53
BC00686=358204,818181,53
BC00687=357648,797481,53
BC00688=358141,799878,53
BC00689=358141,799878,53
BC00690=357648,824051,53
BC00691=357648,824051,53
BC00692=358141,799878,53
BC00693=358141,799878,53
BC00694=358112,801300,53
BC00695=398031,754409,53
BC00696=398031,754409,53
BC00697=279723,674841,53
BC00698=98543,674842,50
BC00699=98543,674842,50
BC00700=164600,674842,50
BC00701=164600,674842,50
BC00702=164600,674842,50
BC00703=164600,674842,50
BC00704=164600,674842,50
BC00705=164600,674842,48
BC00706=164600,674842,48
BC00707=164600,674842,48
BC00708=164600,699931,48
BC00709=164600,699931,48
BC00710=164600,699931,48
BC00711=164600,699931,48
BC00712=164600,699931,48
BC00713=164600,699931,48
BC00714=279723,688848,53
EC00000=797528,-1134
EC00001=797528,-1134
EC00002=798156,0
EC00003=798156,0
EC00004=798156,0
EC00005=798156,0
EC00006=798156,0
EC00007=798156,0
EC00008=798156,0
EC00009=798156,0
EC00010=798156,0
EC00011=798156,0
EC00012=798156,0
EC00013=798156,0
EC00014=798156,0
EC00015=798156,0
EC00016=798156,0
EC00017=798156,0
EC00018=798156,0
EC00019=798156,0
EC00020=798156,0
EC00021=798155,0
EC00022=798155,0
EC00023=798155,0
EC00024=798155,0
EC00025=798155,0
EC00026=798156,0
EC00027=798156,0
EC00028=798156,0
EC00029=798156,0
EC00030=798156,0
EC00031=798156,0
EC00032=798156,0
EC00033=798156,0
EC00034=798156,0
EC00035=798156,0
EC00036=798156,0
EC00037=798156,0
EC00038=798156,0
EC00039=798156,0
EC00040=798156,0
EC00041=798156,0
EC00042=798156,0
EC00043=798156,0
EC00044=798156,0
EC00045=798156,0
EC00046=798156,0
EC00047=798156,0
EC00048=798156,0
EC00049=798156,0
EC00050=798156,0
EC00051=798156,0
EC00052=798156,0
EC00053=798156,0
EC00054=798156,0
EC00055=798156,0
EC00056=798156,0
EC00057=798156,0
EC00058=798156,0
EC00059=798156,0
EC00060=798156,0
EC00061=798156,0
EC00062=798156,0
EC00063=798156,0
EC00064=798156,0
EC00065=798155,1
EC00066=798154,1
EC00067=798154,1
EC00068=798154,1
EC00069=798154,1
EC00070=798154,1
EC00071=798154,1
EC00072=798154,1
EC00073=798154,1
EC00074=798154,1
EC00075=798154,1
EC00076=798154,1
EC00077=798154,1
EC00078=798154,1
EC00079=798154,1
EC00080=798154,1
EC00081=798154,1
EC00082=798154,1
EC00083=798154,1
EC00084=798154,1
EC00085=798154,1
EC00086=798154,1
EC00087=798154,1
EC00088=798154,1
EC00089=798154,1
EC00090=798154,1
EC00091=798154,1
EC00092=798154,1
EC00093=798154,1
EC00094=798154,1
EC00095=798153,1
EC00096=798153,1
EC00097=798153,1
EC00098=798153,1
EC00099=798154,2
EC00100=798153,2
EC00101=798153,2
EC00102=798153,2
EC00103=798153,2
EC00104=798153,2
EC00105=798153,2
EC00106=798153,2
EC00107=798153,2
EC00108=798153,2
EC00109=798153,2
EC00110=798153,2
EC00111=798153,2
EC00112=798153,2
EC00113=798153,2
EC00114=798153,2
EC00115=798155,1
EC00116=798156,0
EC00117=798156,0
EC00118=798156,0
EC00119=798156,0
EC00120=798156,0
EC00121=798156,0
EC00122=798156,0
EC00123=798156,0
EC00124=798156,0
EC00125=798156,0
EC00126=798156,0
EC00127=798154,0
EC00128=798154,0
EC00129=798154,0
EC00130=798154,0
EC00131=798154,0
EC00132=798156,0
EC00133=798156,0
EC00134=798156,0
EC00135=798156,0
EC00136=798156,0
EC00137=798156,0
EC00138=798156,0
EC00139=798156,0
EC00140=798156,0
EC00141=798156,0
EC00142=798156,0
EC00143=798155,0
EC00144=798156,0
EC00145=798156,0
EC00146=798156,0
EC00147=798156,0
EC00148=798156,0
EC00149=798156,0
EC00150=798156,0
EC00151=798156,0
EC00152=798156,0
EC00153=798156,0
EC00154=798156,0
EC00155=798156,0
EC00156=798156,0
EC00157=798156,0
EC00158=798156,0
EC00159=798156,0
EC00160=798156,0
EC00161=798156,0
EC00162=798156,0
EC00163=798156,0
EC00164=798156,0
EC00165=798156,0
EC00166=798156,0
EC00167=798156,0
EC00168=798156,0
EC00169=798156,0
EC00170=798156,0
EC00171=798156,0
EC00172=798156,0
EC00173=798156,0
EC00174=798156,0
EC00175=798156,0
EC00176=798156,0
EC00177=798156,0
EC00178=798156,0
EC00179=798156,0
EC00180=798155,0
EC00181=798156,0
EC00182=798156,0
EC00183=798156,0
EC00184=798156,0
EC00185=798156,0
EC00186=798156,0
EC00187=798156,0
EC00188=798156,0
EC00189=798156,0
EC00190=798156,0
EC00191=798156,0
EC00192=798156,0
EC00193=798156,0
EC00194=798156,0
EC00195=798156,0
EC00196=798156,0
EC00197=798156,0
EC00198=798156,0
EC00199=798156,0
EC00200=798156,0
EC00201=798156,0
EC00202=798156,0
EC00203=798156,0
EC00204=798156,0
EC00205=798156,0
EC00206=798156,0
EC00207=798156,0
EC00208=798156,0
EC00209=798156,0
EC00210=798156,0
EC00211=798156,0
EC00212=798156,0
EC00213=798156,0
EC00214=798156,0
EC00215=798156,0
EC00216=798156,0
EC00217=798156,0
EC00218=798156,0
EC00219=798156,0
EC00220=798156,0
EC00221=798156,0
EC00222=798156,0
EC00223=798156,0
EC00224=798156,0
EC00225=798156,0
EC00226=798156,0
EC00227=798156,0
EC00228=798156,0
EC00229=798156,0
EC00230=798156,0
EC00231=798156,0
EC00232=798156,0
EC00233=798156,0
EC00234=798156,0
EC00235=798156,0
EC00236=798156,0
EC00237=798156,0
EC00238=798156,0
EC00239=798156,0
EC00240=798156,0
EC00241=798156,0
EC00242=798156,0
EC00243=798156,0
EC00244=798156,0
EC00245=798156,0
EC00246=798156,0
EC00247=798156,0
EC00248=798156,0
EC00249=798156,0
EC00250=798156,0
EC00251=798156,0
EC00252=798156,0
EC00253=798156,0
EC00254=798156,0
EC00255=798156,0
EC00256=798156,0
EC00257=798155,0
EC00258=798155,0
EC00259=798155,0
EC00260=798155,0
EC00261=798155,0
EC00262=798155,0
EC00263=798155,0
EC00264=798155,0
EC00265=798155,0
EC00266=798155,0
EC00267=798155,0
EC00268=798155,0
EC00269=798155,0
EC00270=798155,0
EC00271=798155,0
EC00272=798155,0
EC00273=798155,0
EC00274=798155,0
EC00275=798155,0
EC00276=798155,0
EC00277=798154,0
EC00278=798154,0
EC00279=798155,0
EC00280=798155,0
EC00281=798156,0
EC00282=798156,0
EC00283=798156,0
EC00284=798156,0
EC00285=798156,0
EC00286=798156,0
EC00287=798156,0
EC00288=798156,0
EC00289=798156,0
EC00290=798156,0
EC00291=798156,0
EC00292=798156,0
EC00293=798154,0
EC00294=798156,0
EC00295=798156,0
EC00296=798156,0
EC00297=798156,0
EC00298=798156,0
EC00299=798156,0
EC00300=798156,0
EC00301=798156,0
EC00302=798156,0
EC00303=798156,0
EC00304=975524,0
EC00305=975524,0
EC00306=798156,0
EC00307=798156,0
EC00308=798156,0
EC00309=798155,0
EC00310=975524,0
EC00311=975524,0
EC00312=798153,0
EC00313=798156,0
EC00314=798156,0
EC00315=975524,0
EC00316=975524,0
EC00317=798156,0
EC00318=798156,0
EC00319=798156,0
EC00320=798156,0
EC00321=798156,0
EC00322=975524,0
EC00323=975524,0
EC00324=798156,0
EC00325=798156,0
EC00326=798156,0
EC00327=798156,0
EC00328=798156,0
EC00329=798156,0
EC00330=798156,0
EC00331=798156,0
EC00332=798156,0
EC00333=975524,0
EC00334=975524,0
EC00335=798156,0
EC00336=798156,0
EC00337=798156,0
EC00338=798156,0
EC00339=798156,0
EC00340=798156,0
EC00341=798155,1
EC00342=798156,0
EC00343=798156,0
EC00344=798155,1
EC00345=798156,0
EC00346=798156,0
EC00347=798156,0
EC00348=798156,0
EC00349=798156,0
EC00350=798156,0
EC00351=798156,0
EC00352=798156,0
EC00353=798155,0
EC00354=798155,0
EC00355=798156,0
EC00356=798156,0
EC00357=798156,0
EC00358=798156,0
EC00359=798156,0
EC00360=798156,0
EC00361=798156,0
EC00362=798156,0
EC00363=798156,0
EC00364=798156,0
EC00365=798156,0
EC00366=798156,0
EC00367=798156,0
EC00368=798156,0
EC00369=798156,0
EC00370=798156,0
EC00371=798156,0
EC00372=798156,0
EC00373=798156,0
EC00374=798156,0
EC00375=798156,0
EC00376=798156,0
EC00377=798156,0
EC00378=798156,0
EC00379=798156,0
EC00380=798156,0
EC00381=798156,0
EC00382=798156,0
EC00383=798155,0
EC00384=798156,0
EC00385=798156,0
EC00386=798156,0
EC00387=798156,0
EC00388=798153,1
EC00389=798153,1
EC00390=798156,0
EC00391=798156,0
EC00392=798156,0
EC00393=798156,0
EC00394=798156,0
EC00395=798156,0
EC00396=798156,0
EC00397=798156,0
EC00398=798156,0
EC00399=798156,0
EC00400=798156,0
EC00401=798156,0
EC00402=798156,0
EC00403=798156,0
EC00404=798156,0
EC00405=798156,0
EC00406=798156,0
EC00407=798156,0
EC00408=798156,0
EC00409=798156,0
EC00410=798156,0
EC00411=798156,0
EC00412=798156,0
EC00413=798156,0
EC00414=798156,0
EC00415=798156,0
EC00416=798156,0
EC00417=798156,0
EC00418=798156,0
EC00419=798156,0
EC00420=798156,0
EC00421=798156,0
EC00422=798156,0
EC00423=798156,0
EC00424=798156,0
EC00425=798156,0
EC00426=798156,0
EC00427=975524,0
EC00428=975524,0
EC00429=798156,0
EC00430=798156,0
EC00431=798154,1
EC00432=798154,1
EC00433=975524,0
EC00434=975524,0
EC00435=798154,1
EC00436=798154,1
EC00437=798154,1
EC00438=975524,0
EC00439=975524,0
EC00440=975524,0
EC00441=975524,0
EC00442=975524,0
EC00443=975524,0
EC00444=975524,0
EC00445=975524,0
EC00446=975524,0
EC00447=975524,0
EC00448=798670,1
EC00449=800023,0
EC00450=798156,0
EC00451=798156,0
EC00452=798156,0
EC00453=798156,0
EC00454=798156,0
EC00455=798156,0
EC00456=798156,0
EC00457=798156,0
EC00458=798156,0
EC00459=798156,0
EC00460=798156,0
EC00461=798156,0
EC00462=798156,0
EC00463=798156,0
EC00464=798156,0
EC00465=798156,0
EC00466=798156,0
EC00467=798156,0
EC00468=798156,0
EC00469=798156,0
EC00470=798156,0
EC00471=798156,0
EC00472=798156,0
EC00473=798156,0
EC00474=798156,0
EC00475=798156,0
EC00476=798156,0
EC00477=798156,0
EC00478=798156,0
EC00479=798156,0
EC00480=798156,0
EC00481=798155,0
EC00482=798156,0
EC00483=798156,0
EC00484=798156,0
EC00485=798156,0
EC00486=798156,0
EC00487=798156,0
EC00488=798156,0
EC00489=798156,0
EC00490=798156,0
EC00491=798156,0
EC00492=798156,0
EC00493=798156,0
EC00494=798156,0
EC00495=798156,0
EC00496=798156,0
EC00497=798156,0
EC00498=798156,0
EC00499=798156,0
EC00500=798156,0
EC00501=798156,0
EC00502=798156,0
EC00503=798156,0
EC00504=798156,0
EC00505=798156,0
EC00506=798156,0
EC00507=798156,0
EC00508=798154,0
EC00509=798156,0
EC00510=798156,0
EC00511=798156,0
EC00512=798156,0
EC00513=798156,0
EC00514=798156,0
EC00515=798156,0
EC00516=798156,0
EC00517=798156,0
EC00518=798156,0
EC00519=798156,0
EC00520=798156,0
EC00521=798156,0
EC00522=798156,0
EC00523=798156,0
EC00524=798156,0
EC00525=798156,0
EC00526=798156,0
EC00527=798156,0
EC00528=798156,0
EC00529=798156,0
EC00530=798156,0
EC00531=798156,0
EC00532=798156,0
EC00533=798156,0
EC00534=798156,0
EC00535=798156,0
EC00536=798156,0
EC00537=798156,0
EC00538=798156,0
EC00539=798156,0
EC00540=798156,0
EC00541=798156,0
EC00542=798156,0
EC00543=798156,0
EC00544=798156,0
EC00545=798155,1
EC00546=798155,1
EC00547=798155,1
EC00548=798155,1
EC00549=798155,1
EC00550=798154,1
EC00551=798155,1
EC00552=798155,1
EC00553=798155,1
EC00554=798155,1
EC00555=798155,1
EC00556=798155,1
EC00557=798155,1
EC00558=798155,1
EC00559=798155,1
EC00560=798155,1
EC00561=798155,1
EC00562=798155,1
EC00563=798155,1
EC00564=798155,1
EC00565=798155,1
EC00566=798155,1
EC00567=798156,0
EC00568=798156,0
EC00569=798154,1
EC00570=798154,1
EC00571=798154,1
EC00572=798154,1
EC00573=798154,1
EC00574=798154,1
EC00575=798154,1
EC00576=798154,1
EC00577=798156,0
EC00578=798156,0
EC00579=798153,1
EC00580=798153,1
EC00581=798156,0
EC00582=798156,0
EC00583=798153,1
EC00584=798153,1
EC00585=798153,1
EC00586=798156,0
EC00587=798155,1
EC00588=798155,1
EC00589=798154,0
EC00590=798154,0
EC00591=798154,0
EC00592=798154,0
EC00593=798156,0
EC00594=798156,0
EC00595=798154,0
EC00596=798154,0
EC00597=798154,0
EC00598=798156,0
EC00599=798156,0
EC00600=798156,0
EC00601=798156,0
EC00602=798156,0
EC00603=798156,0
EC00604=798156,0
EC00605=798156,0
EC00606=798156,0
EC00607=798156,0
EC00608=798156,0
EC00609=798156,0
EC00610=798156,0
EC00611=798156,0
EC00612=798156,0
EC00613=798156,0
EC00614=798156,0
EC00615=798156,0
EC00616=798156,0
EC00617=798156,0
EC00618=798156,0
EC00619=798156,0
EC00620=798156,0
EC00621=798156,0
EC00622=798154,0
EC00623=798154,0
EC00624=798154,0
EC00625=798156,0
EC00626=798156,0
EC00627=798154,0
EC00628=798154,0
EC00629=798154,0
EC00630=798154,0
EC00631=798154,0
EC00632=798154,0
EC00633=798156,0
EC00634=798156,0
EC00635=798154,0
EC00636=798154,0
EC00637=798154,0
EC00638=798155,0
EC00639=798156,0
EC00640=798156,0
EC00641=798156,0
EC00642=798156,0
EC00643=798156,0
EC00644=798156,0
EC00645=798156,0
EC00646=798156,0
EC00647=798156,0
EC00648=798156,0
EC00649=798156,0
EC00650=798156,0
EC00651=798156,0
EC00652=798156,0
EC00653=798156,0
EC00654=798156,0
EC00655=798156,0
EC00656=798156,0
EC00657=798156,0
EC00658=798156,0
EC00659=798156,0
EC00660=798156,0
EC00661=798156,0
EC00662=798156,0
EC00663=798156,0
EC00664=798156,0
EC00665=798155,0
EC00666=798155,0
EC00667=798156,0
EC00668=798156,0
EC00669=798155,0
EC00670=798155,0
EC00671=798155,0
EC00672=798155,0
EC00673=798155,0
EC00674=798156,0
EC00675=798156,0
EC00676=798156,0
EC00677=798156,0
EC00678=798156,0
EC00679=798156,0
EC00680=798156,0
EC00681=798156,0
EC00682=798156,0
EC00683=798156,0
EC00684=798156,0
EC00685=798156,0
EC00686=798156,0
EC00687=798156,0
EC00688=798156,0
EC00689=798156,0
EC00690=798156,0
EC00691=798156,0
EC00692=798156,0
EC00693=798156,0
EC00694=798156,0
EC00695=798156,0
EC00696=798156,0
EC00697=798156,0
EC00698=798155,1
EC00699=798155,1
EC00700=798155,1
EC00701=798155,1
EC00702=798155,1
EC00703=798155,1
EC00704=798155,1
EC00705=798153,1
EC00706=798153,1
EC00707=798153,1
EC00708=798153,1
EC00709=798153,1
EC00710=798153,1
EC00711=798153,1
EC00712=798153,1
EC00713=798153,1
EC00714=798156,0
///POSTYPE BASE
///RECTAN
///RCONF 0,0,0,0,0,0,0,0,0,0,0,0,0,0,0,0,0,0,0,0,0,0,0,0
P00006=0.222,-3.123,-1.508,0.0000,0.0000,0.0000
P00021=-0.225,-6.128,-0.405,0.0000,0.0000,0.0000
P00022=0.222,-3.123,-1.508,0.0000,0.0000,0.0000
P00023=0.143,-0.036,0.682,0.0000,0.0000,0.0000
P00030=5.926,-4.294,-1.390,0.0000,0.0000,0.0000
P00031=1.853,-0.001,-1.549,0.0000,0.0000,0.0000
P00032=1.957,0.503,-7.217,0.0000,0.0000,0.0000
///RCONF 0,0,0,0,1,0,0,0,0,0,0,0,0,0,0,0,0,0,0,0,0,0,0,0
P00033=-0.123,0.612,-5.012,0.0000,0.0000,0.0000
///RCONF 0,0,0,0,0,0,0,0,0,0,0,0,0,0,0,0,0,0,0,0,0,0,0,0
P00034=-0.304,0.773,-2.693,0.0000,0.0000,0.0000
P00035=2.817,0.591,-1.622,0.0000,0.0000,0.0000
P00036=-1.108,-0.829,1.850,0.0000,0.0000,0.0000
P00037=0.023,0.937,-2.677,0.0000,0.0000,0.0000
P00038=0.158,-1.133,-1.952,0.0000,0.0000,0.0000
P00039=0.012,-3.081,-0.106,0.0000,0.0000,0.0000
P00040=-0.030,9.648,2.467,0.0000,0.0000,0.0000
P00041=0.192,3.924,0.305,0.0000,0.0000,0.0000
P00042=-0.217,1.941,0.413,0.0000,0.0000,0.0000
P00050=4.296,-4.501,-0.826,0.0000,0.0000,0.0000
P00052=0.088,2.832,-0.342,0.0000,0.0000,0.0000
P00055=-0.342,8.912,1.324,0.0000,0.0000,0.0000
P00056=0.568,-0.032,0.830,0.0000,0.0000,0.0000
P00057=0.586,-0.180,1.727,0.0000,0.0000,0.0000
P00058=0.385,-0.061,1.027,0.0000,0.0000,0.0000
P00060=2.327,-2.514,-2.692,0.0000,0.0000,0.0000
P00061=1.575,-3.405,-0.752,0.0000,0.0000,0.0000
P00062=-0.135,-0.848,-1.706,0.0000,0.0000,0.0000
P00063=0.036,-0.654,-3.005,0.0000,0.0000,0.0000
P00064=-0.056,-0.423,-1.596,0.0000,0.0000,0.0000
P00090=0.184,3.539,2.293,0.0000,0.0000,0.0000
P00091=-0.109,0.052,-0.075,0.0000,0.0000,0.0000
//INST
///DATE 2025/04/22 13:19
///ATTR SC,RW
///GROUP1 RB1,BS1
///GROUP2 ST1
NOP
'OK_r2_O8A-O21A(90,0)
'Path S1018
MOVJ C00000 BC00000 VJ=50.00  +MOVJ EC00000 VJ=10.00
MOVJ C00001 BC00001 VJ=100.00  +MOVJ EC00001 VJ=100.00
SFTOF3D
MOVJ C00002 BC00002 VJ=100.00  +MOVJ EC00002 VJ=100.00
MOVL C00003 BC00003 V=400.0  +MOVJ EC00003 VJ=100.00
SMOVL C00004 BC00004 V=100.0  +MOVJ EC00004
SREFP 3 C00005 BC00005  +REFP EC00005
CALL JOB:SEARCH-R1-S13D
SET P031 P006
SFTON3D P031
SMOVL C00006 BC00006 V=100.0  +MOVJ EC00006
SREFP 3 C00007 BC00007  +REFP EC00007
CALL JOB:SEARCH-R1-S13D
SET P031 P006
SFTON3D P031
SFTOF3D
SMOVL C00008 BC00008 V=100.0  +MOVJ EC00008
MOVL C00009 BC00009 V=400.0  +MOVJ EC00009 VJ=100.00
SMOVL C00010 BC00010 V=100.0  +MOVJ EC00010
SREFP 3 C00011 BC00011  +REFP EC00011
CALL JOB:SEARCH-R1-S13D
SET P064 P006
SFTON3D P064
SMOVL C00012 BC00012 V=100.0  +MOVJ EC00012
SREFP 3 C00013 BC00013  +REFP EC00013
CALL JOB:SEARCH-R1-S13D
SET P064 P006
SFTON3D P064
SMOVL C00014 BC00014 V=100.0  +MOVJ EC00014
SMOVL C00015 BC00015 V=100.0  +MOVJ EC00015
SREFP 3 C00016 BC00016  +REFP EC00016
CALL JOB:SEARCH-R1-S13D
SET P061 P006
SFTON3D P061
SMOVL C00017 BC00017 V=100.0  +MOVJ EC00017
SFTOF3D
SMOVL C00018 BC00018 V=100.0  +MOVJ EC00018
SMOVL C00019 BC00019 V=333.3  +MOVJ EC00019
MOVL C00020 BC00020 V=333.3  +MOVJ EC00020 VJ=100.00
SMOVL C00021 BC00021 V=100.0  +MOVJ EC00021
SREFP 3 C00022 BC00022  +REFP EC00022
CALL JOB:SEARCH-R1-S13D
SET P032 P006
SFTON3D P032
SMOVL C00023 BC00023 V=100.0  +MOVJ EC00023
SREFP 3 C00024 BC00024  +REFP EC00024
CALL JOB:SEARCH-R1-S13D
SET P032 P006
SFTON3D P032
SMOVL C00025 BC00025 V=250.0  +MOVJ EC00025
MOVL C00026 BC00026 V=1000.0  +MOVJ EC00026 VJ=100.00
'Path S1554
SFTOF3D
MOVJ C00027 BC00027 VJ=100.00  +MOVJ EC00027 VJ=100.00
MOVL C00028 BC00028 V=400.0  +MOVJ EC00028 VJ=100.00
SMOVL C00029 BC00029 V=100.0  +MOVJ EC00029
SMOVL C00030 BC00030 V=100.0  +MOVJ EC00030
SREFP 3 C00031 BC00031  +REFP EC00031
CALL JOB:SEARCH-R1-S13D
SET P035 P006
SFTON3D P035
SMOVL C00032 BC00032 V=100.0  +MOVJ EC00032
SMOVL C00033 BC00033 V=100.0  +MOVJ EC00033
SMOVL C00034 BC00034 V=100.0  +MOVJ EC00034
SREFP 3 C00035 BC00035  +REFP EC00035
CALL JOB:SEARCH-R1-S13D
SET P035 P006
SFTON3D P035
SMOVL C00036 BC00036 V=166.7  +MOVJ EC00036
MOVL C00037 BC00037 V=1000.0  +MOVJ EC00037 VJ=100.00
MOVJ C00038 BC00038 VJ=50.00  +MOVJ EC00038 VJ=10.00
MOVJ C00039 BC00039 VJ=100.00  +MOVJ EC00039 VJ=100.00
'Path S1019
SFTOF3D
MOVJ C00040 BC00040 VJ=100.00  +MOVJ EC00040 VJ=100.00
MOVL C00041 BC00041 V=400.0  +MOVJ EC00041 VJ=100.00
SMOVL C00042 BC00042 V=100.0  +MOVJ EC00042
SREFP 3 C00043 BC00043  +REFP EC00043
CALL JOB:SEARCH-R1-S13D
SET P050 P006
SFTON3D P050
SMOVL C00044 BC00044 V=100.0  +MOVJ EC00044
SREFP 3 C00045 BC00045  +REFP EC00045
CALL JOB:SEARCH-R1-S13D
SET P050 P006
SFTON3D P050
SMOVL C00046 BC00046 V=166.7  +MOVJ EC00046
SMOVL C00047 BC00047 V=166.7  +MOVJ EC00047
SREFP 3 C00048 BC00048  +REFP EC00048
CALL JOB:SEARCH-R1-S13D
SET P050 P006
SFTON3D P050
SMOVL C00049 BC00049 V=166.7  +MOVJ EC00049
MOVL C00050 BC00050 V=1000.0  +MOVJ EC00050 VJ=100.00
MOVJ C00051 BC00051 VJ=100.00  +MOVJ EC00051 VJ=100.00
'OBROT 110
MOVJ C00052 BC00052 VJ=100.00  +MOVJ EC00052 VJ=100.00
MOVJ C00053 BC00053 VJ=100.00  +MOVJ EC00053 VJ=100.00
MOVJ C00054 BC00054 VJ=100.00  +MOVJ EC00054 VJ=100.00
'Path S1020
SFTOF3D
SMOVL C00055 BC00055 V=166.7  +MOVJ EC00055
SREFP 3 C00056 BC00056  +REFP EC00056
CALL JOB:SEARCH-R1-S13D
SET P033 P006
SFTON3D P033
SMOVL C00057 BC00057 V=166.7  +MOVJ EC00057
SREFP 3 C00058 BC00058  +REFP EC00058
CALL JOB:SEARCH-R1-S13D
SET P033 P006
SFTON3D P033
MOVJ C00059 BC00059 VJ=50.00  +MOVJ EC00059 VJ=50.00
MOVJ C00060 BC00060 VJ=50.00  +MOVJ EC00060 VJ=100.00
SMOVL C00061 BC00061 V=100.0  +MOVJ EC00061
SREFP 3 C00062 BC00062  +REFP EC00062
CALL JOB:SEARCH-R1-S13D
SET P033 P006
SFTON3D P033
SMOVL C00063 BC00063 V=166.7  +MOVJ EC00063
MOVL C00064 BC00064 V=666.7  +MOVJ EC00064 VJ=100.00
MOVJ C00065 BC00065 VJ=50.00  +MOVJ EC00065 VJ=50.00
MOVJ C00066 BC00066 VJ=50.00  +MOVJ EC00066 VJ=50.00
MOVJ C00067 BC00067 VJ=50.00  +MOVJ EC00067 VJ=50.00
'Path S1025
SFTOF3D
SMOVL C00068 BC00068 V=60.0  +MOVJ EC00068
SREFP 3 C00069 BC00069  +REFP EC00069
CALL JOB:SEARCH-R1-S13D
SET P038 P006
SFTON3D P038
SMOVL C00070 BC00070 V=100.0  +MOVJ EC00070
SREFP 3 C00071 BC00071  +REFP EC00071
CALL JOB:SEARCH-R1-S13D
SET P038 P006
SFTON3D P038
SMOVL C00072 BC00072 V=100.0  +MOVJ EC00072
SMOVL C00073 BC00073 V=166.7  +MOVJ EC00073
MOVJ C00074 BC00074 VJ=100.00  +MOVJ EC00074 VJ=15.00
MOVJ C00075 BC00075 VJ=100.00  +MOVJ EC00075 VJ=50.00
MOVJ C00076 BC00076 VJ=100.00  +MOVJ EC00076 VJ=15.00
MOVJ C00077 BC00077 VJ=15.00  +MOVJ EC00077 VJ=50.00
SMOVL C00078 BC00078 V=100.0  +MOVJ EC00078
SREFP 3 C00079 BC00079  +REFP EC00079
CALL JOB:SEARCH-R1-S13D
SET P038 P006
SFTON3D P038
SMOVL C00080 BC00080 V=100.0  +MOVJ EC00080
MOVJ C00081 BC00081 VJ=100.00  +MOVJ EC00081 VJ=15.00
MOVL C00082 BC00082 V=833.3  +MOVJ EC00082 VJ=100.00
MOVJ C00083 BC00083 VJ=100.00  +MOVJ EC00083 VJ=15.00
MOVJ C00084 BC00084 VJ=100.00  +MOVJ EC00084 VJ=15.00
'Path S1027
SFTOF3D
MOVL C00085 BC00085 V=400.0  +MOVJ EC00085 VJ=100.00
SMOVL C00086 BC00086 V=100.0  +MOVJ EC00086
SREFP 3 C00087 BC00087  +REFP EC00087
CALL JOB:SEARCH-R1-S13D
SET P040 P006
SFTON3D P040
SMOVL C00088 BC00088 V=100.0  +MOVJ EC00088
SMOVL C00089 BC00089 V=133.3  +MOVJ EC00089
SMOVL C00090 BC00090 V=100.0  +MOVJ EC00090
SREFP 3 C00091 BC00091  +REFP EC00091
CALL JOB:SEARCH-R1-S13D
SET P040 P006
SFTON3D P040
SMOVL C00092 BC00092 V=133.3  +MOVJ EC00092
MOVJ C00093 BC00093 VJ=100.00  +MOVJ EC00093 VJ=15.00
MOVJ C00094 BC00094 VJ=100.00  +MOVJ EC00094 VJ=15.00
SMOVL C00095 BC00095 V=100.0  +MOVJ EC00095
SREFP 3 C00096 BC00096  +REFP EC00096
CALL JOB:SEARCH-R1-S13D
SET P040 P006
SFTON3D P040
SMOVL C00097 BC00097 V=100.0  +MOVJ EC00097
'Path S1023
SFTOF3D
MOVJ C00098 BC00098 VJ=100.00  +MOVJ EC00098 VJ=15.00
MOVJ C00099 BC00099 VJ=50.00  +MOVJ EC00099 VJ=15.00
MOVJ C00100 BC00100 VJ=50.00  +MOVJ EC00100 VJ=15.00
MOVJ C00101 BC00101 VJ=50.00  +MOVJ EC00101 VJ=15.00
SMOVL C00102 BC00102 V=100.0  +MOVJ EC00102
SREFP 3 C00103 BC00103  +REFP EC00103
CALL JOB:SEARCH-R1-S13D
SET P036 P006
SFTON3D P036
SMOVL C00104 BC00104 V=100.0  +MOVJ EC00104
SREFP 3 C00105 BC00105  +REFP EC00105
CALL JOB:SEARCH-R1-S13D
SET P036 P006
SFTON3D P036
SMOVL C00106 BC00106 V=100.0  +MOVJ EC00106
SMOVL C00107 BC00107 V=133.3  +MOVJ EC00107
SMOVL C00108 BC00108 V=100.0  +MOVJ EC00108
SREFP 3 C00109 BC00109  +REFP EC00109
CALL JOB:SEARCH-R1-S13D
SET P036 P006
SFTON3D P036
SMOVL C00110 BC00110 V=100.0  +MOVJ EC00110
SMOVL C00111 BC00111 V=250.0  +MOVJ EC00111
SMOVL C00112 BC00112 V=833.3  +MOVJ EC00112
MOVJ C00113 BC00113 VJ=100.00  +MOVJ EC00113 VJ=15.00
MOVJ C00114 BC00114 VJ=100.00  +MOVJ EC00114 VJ=15.00
MOVJ C00115 BC00115 VJ=100.00  +MOVJ EC00115 VJ=15.00
'Path S1024
SFTOF3D
MOVJ C00116 BC00116 VJ=100.00  +MOVJ EC00116 VJ=100.00
MOVL C00117 BC00117 V=400.0  +MOVJ EC00117 VJ=100.00
SMOVL C00118 BC00118 V=100.0  +MOVJ EC00118
SREFP 3 C00119 BC00119  +REFP EC00119
CALL JOB:SEARCH-R1-S13D
SET P037 P006
SFTON3D P037
SMOVL C00120 BC00120 V=100.0  +MOVJ EC00120
SREFP 3 C00121 BC00121  +REFP EC00121
CALL JOB:SEARCH-R1-S13D
SET P037 P006
SFTON3D P037
SMOVL C00122 BC00122 V=100.0  +MOVJ EC00122
MOVL C00123 BC00123 V=400.0  +MOVJ EC00123 VJ=100.00
MOVL C00124 BC00124 V=1000.0  +MOVJ EC00124 VJ=100.00
MOVJ C00125 BC00125 VJ=100.00  +MOVJ EC00125 VJ=100.00
'Path S1028
SFTOF3D
MOVJ C00126 BC00126 VJ=100.00  +MOVJ EC00126 VJ=100.00
SMOVL C00127 BC00127 V=100.0  +MOVJ EC00127
SREFP 3 C00128 BC00128  +REFP EC00128
CALL JOB:SEARCH-R1-S13D
SET P041 P006
SFTON3D P041
SMOVL C00129 BC00129 V=100.0  +MOVJ EC00129
SREFP 3 C00130 BC00130  +REFP EC00130
CALL JOB:SEARCH-R1-S13D
SET P041 P006
SFTON3D P041
SFTOF3D
SMOVL C00131 BC00131 V=100.0  +MOVJ EC00131
MOVL C00132 BC00132 V=400.0  +MOVJ EC00132 VJ=100.00
MOVL C00133 BC00133 V=400.0  +MOVJ EC00133 VJ=15.00
SMOVL C00134 BC00134 V=100.0  +MOVJ EC00134
SREFP 3 C00135 BC00135  +REFP EC00135
CALL JOB:SEARCH-R1-S13D
SET P042 P006
SFTON3D P042
SMOVL C00136 BC00136 V=100.0  +MOVJ EC00136
SREFP 3 C00137 BC00137  +REFP EC00137
CALL JOB:SEARCH-R1-S13D
SET P042 P006
SFTON3D P042
SMOVL C00138 BC00138 V=100.0  +MOVJ EC00138
SFTOF3D
SMOVL C00139 BC00139 V=333.3  +MOVJ EC00139
SMOVL C00140 BC00140 V=100.0  +MOVJ EC00140
SREFP 3 C00141 BC00141  +REFP EC00141
CALL JOB:SEARCH-R1-S13D
SET P062 P006
SFTON3D P062
SMOVL C00142 BC00142 V=100.0  +MOVJ EC00142
SREFP 3 C00143 BC00143  +REFP EC00143
CALL JOB:SEARCH-R1-S13D
SET P062 P006
SFTON3D P062
SMOVL C00144 BC00144 V=100.0  +MOVJ EC00144
SMOVL C00145 BC00145 V=333.3  +MOVJ EC00145
SMOVL C00146 BC00146 V=333.3  +MOVJ EC00146
SMOVL C00147 BC00147 V=100.0  +MOVJ EC00147
SREFP 3 C00148 BC00148  +REFP EC00148
CALL JOB:SEARCH-R1-S13D
SET P063 P006
SFTON3D P063
SMOVL C00149 BC00149 V=100.0  +MOVJ EC00149
SFTOF3D
MOVL C00150 BC00150 V=1000.0  +MOVJ EC00150 VJ=100.00
'Path S1029
MOVJ C00151 BC00151 VJ=100.00  +MOVJ EC00151 VJ=10.00
MOVJ C00152 BC00152 VJ=100.00  +MOVJ EC00152 VJ=10.00
SFTOF3D
MOVJ C00153 BC00153 VJ=100.00  +MOVJ EC00153 VJ=100.00
MOVL C00154 BC00154 V=400.0  +MOVJ EC00154 VJ=100.00
SMOVL C00155 BC00155 V=100.0  +MOVJ EC00155
SREFP 3 C00156 BC00156  +REFP EC00156
CALL JOB:SEARCH-R1-S13D
SET P052 P006
SFTON3D P052
SMOVL C00157 BC00157 V=100.0  +MOVJ EC00157
SMOVL C00158 BC00158 V=100.0  +MOVJ EC00158
SREFP 3 C00159 BC00159  +REFP EC00159
CALL JOB:SEARCH-R1-S13D
SET P052 P006
SFTON3D P052
SMOVL C00160 BC00160 V=133.3  +MOVJ EC00160
MOVL C00161 BC00161 V=400.0  +MOVJ EC00161 VJ=100.00
MOVL C00162 BC00162 V=1000.0  +MOVJ EC00162 VJ=100.00
MOVJ C00163 BC00163 VJ=100.00  +MOVJ EC00163 VJ=10.00
MOVJ C00164 BC00164 VJ=100.00  +MOVJ EC00164 VJ=100.00
MOVL C00165 BC00165 V=1000.0  +MOVJ EC00165 VJ=100.00
SMOVL C00166 BC00166 V=500.0  +MOVJ EC00166
SMOVL C00167 BC00167 V=166.7  +MOVJ EC00167
SREFP 3 C00168 BC00168  +REFP EC00168
CALL JOB:SEARCH-R1-S13D
SET P055 P006
SFTON3D P055
SMOVL C00169 BC00169 V=100.0  +MOVJ EC00169
SREFP 3 C00170 BC00170  +REFP EC00170
CALL JOB:SEARCH-R1-S13D
SET P055 P006
SFTON3D P055
SMOVL C00171 BC00171 V=166.7  +MOVJ EC00171
SFTOF3D
SMOVL C00172 BC00172 V=500.0  +MOVJ EC00172
SMOVL C00173 BC00173 V=166.7  +MOVJ EC00173
SREFP 3 C00174 BC00174  +REFP EC00174
CALL JOB:SEARCH-R1-S13D
SET P060 P006
SFTON3D P060
SMOVL C00175 BC00175 V=100.0  +MOVJ EC00175
SREFP 3 C00176 BC00176  +REFP EC00176
CALL JOB:SEARCH-R1-S13D
SET P060 P006
SFTON3D P060
SMOVL C00177 BC00177 V=166.7  +MOVJ EC00177
SMOVL C00178 BC00178 V=666.7  +MOVJ EC00178
MOVJ C00179 BC00179 VJ=100.00  +MOVJ EC00179 VJ=100.00
'Path S1026
SFTOF3D
MOVJ C00180 BC00180 VJ=100.00  +MOVJ EC00180 VJ=10.00
MOVJ C00181 BC00181 VJ=100.00  +MOVJ EC00181 VJ=100.00
MOVL C00182 BC00182 V=400.0  +MOVJ EC00182 VJ=100.00
SMOVL C00183 BC00183 V=166.7  +MOVJ EC00183
SREFP 3 C00184 BC00184  +REFP EC00184
CALL JOB:SEARCH-R1-S13D
SET P039 P006
SFTON3D P039
SMOVL C00185 BC00185 V=100.0  +MOVJ EC00185
SMOVL C00186 BC00186 V=100.0  +MOVJ EC00186
SREFP 3 C00187 BC00187  +REFP EC00187
CALL JOB:SEARCH-R1-S13D
SET P039 P006
SFTON3D P039
SMOVL C00188 BC00188 V=166.7  +MOVJ EC00188
SMOVL C00189 BC00189 V=333.3  +MOVJ EC00189
SMOVL C00190 BC00190 V=100.0  +MOVJ EC00190
SREFP 3 C00191 BC00191  +REFP EC00191
CALL JOB:SEARCH-R1-S13D
SET P039 P006
SFTON3D P039
SMOVL C00192 BC00192 V=100.0  +MOVJ EC00192
SMOVL C00193 BC00193 V=250.0  +MOVJ EC00193
SMOVL C00194 BC00194 V=166.7  +MOVJ EC00194
MOVL C00195 BC00195 V=400.0  +MOVJ EC00195 VJ=100.00
MOVL C00196 BC00196 V=1000.0  +MOVJ EC00196 VJ=100.00
'Path S1021
SFTOF3D
MOVJ C00197 BC00197 VJ=100.00  +MOVJ EC00197 VJ=100.00
MOVL C00198 BC00198 V=400.0  +MOVJ EC00198 VJ=100.00
SMOVL C00199 BC00199 V=100.0  +MOVJ EC00199
SREFP 3 C00200 BC00200  +REFP EC00200
CALL JOB:SEARCH-R1-S13D
SET P034 P006
SFTON3D P034
SMOVL C00201 BC00201 V=100.0  +MOVJ EC00201
SMOVL C00202 BC00202 V=133.3  +MOVJ EC00202
SMOVL C00203 BC00203 V=100.0  +MOVJ EC00203
SREFP 3 C00204 BC00204  +REFP EC00204
CALL JOB:SEARCH-R1-S13D
SET P034 P006
SFTON3D P034
SMOVL C00205 BC00205 V=100.0  +MOVJ EC00205
SMOVL C00206 BC00206 V=100.0  +MOVJ EC00206
SREFP 3 C00207 BC00207  +REFP EC00207
CALL JOB:SEARCH-R1-S13D
SET P034 P006
SFTON3D P034
SMOVL C00208 BC00208 V=133.3  +MOVJ EC00208
MOVL C00209 BC00209 V=400.0  +MOVJ EC00209 VJ=100.00
MOVL C00210 BC00210 V=1000.0  +MOVJ EC00210 VJ=100.00
MOVJ C00211 BC00211 VJ=100.00  +MOVJ EC00211 VJ=100.00
MOVJ C00212 BC00212 VJ=100.00  +MOVJ EC00212 VJ=100.00
MOVJ C00213 BC00213 VJ=100.00  +MOVJ EC00213 VJ=100.00
SMOVL C00214 BC00214 V=100.0  +MOVJ EC00214
SREFP 3 C00215 BC00215  +REFP EC00215
CALL JOB:SEARCH-R1-S13D
SET P056 P006
SFTON3D P056
SMOVL C00216 BC00216 V=100.0  +MOVJ EC00216
SREFP 3 C00217 BC00217  +REFP EC00217
CALL JOB:SEARCH-R1-S13D
SET P056 P006
SFTON3D P056
SFTOF3D
SMOVL C00218 BC00218 V=100.0  +MOVJ EC00218
SMOVL C00219 BC00219 V=250.0  +MOVJ EC00219
SMOVL C00220 BC00220 V=100.0  +MOVJ EC00220
SREFP 3 C00221 BC00221  +REFP EC00221
CALL JOB:SEARCH-R1-S13D
SET P057 P006
SFTON3D P057
SMOVL C00222 BC00222 V=100.0  +MOVJ EC00222
SREFP 3 C00223 BC00223  +REFP EC00223
CALL JOB:SEARCH-R1-S13D
SET P057 P006
SFTON3D P057
SFTOF3D
SMOVL C00224 BC00224 V=100.0  +MOVJ EC00224
SMOVL C00225 BC00225 V=333.3  +MOVJ EC00225
MOVJ C00226 BC00226 VJ=100.00  +MOVJ EC00226 VJ=100.00
MOVJ C00227 BC00227 VJ=100.00  +MOVJ EC00227 VJ=100.00
MOVJ C00228 BC00228 VJ=100.00  +MOVJ EC00228 VJ=100.00
SMOVL C00229 BC00229 V=166.7  +MOVJ EC00229
SREFP 3 C00230 BC00230  +REFP EC00230
CALL JOB:SEARCH-R1-S13D
SET P058 P006
SFTON3D P058
SMOVL C00231 BC00231 V=166.7  +MOVJ EC00231
SREFP 3 C00232 BC00232  +REFP EC00232
CALL JOB:SEARCH-R1-S13D
SET P058 P006
SFTON3D P058
SFTOF3D
SMOVL C00233 BC00233 V=166.7  +MOVJ EC00233
SMOVL C00234 BC00234 V=666.7  +MOVJ EC00234
MOVJ C00235 BC00235 VJ=100.00  +MOVJ EC00235 VJ=100.00
MOVJ C00236 BC00236 VJ=100.00  +MOVJ EC00236 VJ=100.00
SMOVL C00237 BC00237 V=666.7  +MOVJ EC00237
SMOVL C00238 BC00238 V=166.7  +MOVJ EC00238
SREFP 3 C00239 BC00239  +REFP EC00239
CALL JOB:SEARCH-R1-S13D
SET P090 P006
SFTON3D P090
SMOVL C00240 BC00240 V=166.7  +MOVJ EC00240
SREFP 3 C00241 BC00241  +REFP EC00241
CALL JOB:SEARCH-R1-S13D
SET P090 P006
SFTON3D P090
SFTOF3D
SMOVL C00242 BC00242 V=166.7  +MOVJ EC00242
SMOVL C00243 BC00243 V=500.0  +MOVJ EC00243
SMOVL C00244 BC00244 V=166.7  +MOVJ EC00244
SREFP 3 C00245 BC00245  +REFP EC00245
CALL JOB:SEARCH-R1-S13D
SET P091 P006
SFTON3D P091
SMOVL C00246 BC00246 V=166.7  +MOVJ EC00246
SREFP 3 C00247 BC00247  +REFP EC00247
CALL JOB:SEARCH-R1-S13D
SET P091 P006
SFTON3D P091
SFTOF3D
SMOVL C00248 BC00248 V=166.7  +MOVJ EC00248
MACRO1 MJ#(0) ARGF6
SFTON3D P091
SMOVL C00249 BC00249 V=133.3  +MOVJ EC00249
ARCON
SMOVL C00250 BC00250 V=12.5  +MOVJ EC00250
SFTON3D P090
SMOVL C00251 BC00251 V=12.5  +MOVJ EC00251
ARCOF
SFTOF3D
SMOVL C00252 BC00252 V=166.7  +MOVJ EC00252
SMOVL C00253 BC00253 V=1000.0  +MOVJ EC00253
MOVJ C00254 BC00254 VJ=100.00  +MOVJ EC00254 VJ=100.00
MOVJ C00255 BC00255 VJ=100.00  +MOVJ EC00255 VJ=100.00
MACRO1 MJ#(0) ARGF14
SFTON3D P034
SMOVL C00256 BC00256 V=166.7  +MOVJ EC00256
ARCON
SMOVL C00257 BC00257 V=11.7  +MOVJ EC00257
ARCOF
MOVJ C00258 BC00258 VJ=25.00  +MOVJ EC00258 VJ=100.00
MOVJ C00259 BC00259 VJ=100.00  +MOVJ EC00259 VJ=25.00
SFTON3D P058
SMOVL C00260 BC00260 V=166.7  +MOVJ EC00260
ARCON
SMOVL C00261 BC00261 V=10.0  +MOVJ EC00261
ARCOF
SFTOF3D
SMOVL C00262 BC00262 V=166.7  +MOVJ EC00262
MACRO1 MJ#(0) ARGF9
SMOVL C00263 BC00263 V=500.0  +MOVJ EC00263
SFTON3D P034
SMOVL C00264 BC00264 V=250.0  +MOVJ EC00264
ARCON
SMOVL C00265 BC00265 V=9.2  +MOVJ EC00265
SFTON3D P057
SMOVL C00266 BC00266 V=9.2  +MOVJ EC00266
SMOVL C00267 BC00267 V=9.2  +MOVJ EC00267
SMOVL C00268 BC00268 V=9.2  +MOVJ EC00268
COMM SREFP 1 C00269 BC00269  +REFP EC00269
COMM SREFP 2 C00270 BC00270  +REFP EC00270
SFTON3D P056
COMM SWVON WEV#(30)
SMOVL C00271 BC00271 V=8.7  +MOVJ EC00271
COMM SMOVL C00272 BC00272 V=8.7  +MOVJ EC00272
SMOVL C00273 BC00273 V=8.7  +MOVJ EC00273
ARCOF
SFTOF3D
SMOVL C00274 BC00274 V=333.3  +MOVJ EC00274
MOVJ C00275 BC00275 VJ=100.00  +MOVJ EC00275 VJ=25.00
MOVJ C00276 BC00276 VJ=100.00  +MOVJ EC00276 VJ=25.00
SFTON3D P057
SMOVL C00277 BC00277 V=166.7  +MOVJ EC00277
ARCON
COMM SWVON WEV#(30)
SMOVL C00278 BC00278 V=9.2  +MOVJ EC00278
ARCOF
SWVOF
SFTOF3D
SMOVL C00279 BC00279 V=166.7  +MOVJ EC00279
MOVJ C00280 BC00280 VJ=100.00  +MOVJ EC00280 VJ=25.00
'
MOVJ C00281 BC00281 VJ=100.00  +MOVJ EC00281 VJ=100.00
'Path W939
SFTOF3D
SFTON3D P039
MOVJ C00282 BC00282 VJ=100.00  +MOVJ EC00282 VJ=100.00
SMOVL C00283 BC00283 V=400.0  +MOVJ EC00283
SMOVL C00284 BC00284 V=166.7 PL=0  +MOVJ EC00284
SREFP 1 C00285 BC00285  +REFP EC00285
SREFP 2 C00286 BC00286  +REFP EC00286
MACRO1 MJ#(0) ARGF14
ARCON
SMOVL C00287 BC00287 V=10.0  +MOVJ EC00287
ARCOF
SMOVL C00288 BC00288 V=400.0  +MOVJ EC00288
SMOVL C00289 BC00289 V=1000.0  +MOVJ EC00289
SFTOF3D
MOVJ C00290 BC00290 VJ=100.00  +MOVJ EC00290 VJ=100.00
'Path W941
SFTOF3D
SFTON3D P039
MOVJ C00291 BC00291 VJ=100.00  +MOVJ EC00291 VJ=100.00
SMOVL C00292 BC00292 V=400.0  +MOVJ EC00292
SMOVL C00293 BC00293 V=133.3 PL=0  +MOVJ EC00293
SREFP 1 C00294 BC00294  +REFP EC00294
SREFP 2 C00295 BC00295  +REFP EC00295
ARCON
SMOVL C00296 BC00296 V=10.0  +MOVJ EC00296
ARCOF
SMOVL C00297 BC00297 V=400.0  +MOVJ EC00297
SFTOF3D
SMOVL C00298 BC00298 V=1000.0  +MOVJ EC00298
MOVJ C00299 BC00299 VJ=100.00  +MOVJ EC00299 VJ=10.00
SFTOF3D
MOVJ C00300 BC00300 VJ=100.00  +MOVJ EC00300 VJ=100.00
MOVJ C00301 BC00301 VJ=100.00  +MOVJ EC00301 VJ=15.00
'9
'Path W942
SFTOF3D
SFTON3D P038
COMM MOVJ C00302 BC00302 VJ=100.00  +MOVJ EC00302 VJ=100.00
COMM SMOVL C00303 BC00303 V=166.7 PL=0  +MOVJ EC00303
COMM SREFP 1 C00304 BC00304  +REFP EC00304
COMM SREFP 2 C00305 BC00305  +REFP EC00305
COMM MACRO1 MJ#(0) ARGF14
COMM ARCON
COMM SMOVL C00306 BC00306 V=10.0  +MOVJ EC00306
COMM ARCOF
COMM SFTOF3D
COMM SMOVL C00307 BC00307 V=400.0  +MOVJ EC00307
COMM SMOVL C00308 BC00308 V=1000.0  +MOVJ EC00308
COMM SFTOF3D
COMM 'Path W943
SFTOF3D
SFTON3D P038
SMOVL C00309 BC00309 V=133.3 PL=0  +MOVJ EC00309
SREFP 1 C00310 BC00310  +REFP EC00310
SREFP 2 C00311 BC00311  +REFP EC00311
MACRO1 MJ#(0) ARGF14
ARCON
SMOVL C00312 BC00312 V=10.0  +MOVJ EC00312
ARCOF
SMOVL C00313 BC00313 V=400.0  +MOVJ EC00313
SFTOF3D
'Path W944
SFTOF3D
SFTON3D P038
SMOVL C00314 BC00314 V=166.7 PL=0  +MOVJ EC00314
SREFP 1 C00315 BC00315  +REFP EC00315
SREFP 2 C00316 BC00316  +REFP EC00316
MACRO1 MJ#(0) ARGF14
ARCON
SMOVL C00317 BC00317 V=10.0  +MOVJ EC00317
SMOVL C00318 BC00318 V=10.0  +MOVJ EC00318
ARCOF
SMOVL C00319 BC00319 V=400.0  +MOVJ EC00319
SFTOF3D
'10
'11
MOVJ C00320 BC00320 VJ=100.00  +MOVJ EC00320 VJ=100.00
'Path W946
SFTOF3D
SFTON3D P033
SMOVL C00321 BC00321 V=166.7 PL=0  +MOVJ EC00321
SREFP 1 C00322 BC00322  +REFP EC00322
SREFP 2 C00323 BC00323  +REFP EC00323
MACRO1 MJ#(0) ARGF14
ARCON
SMOVL C00324 BC00324 V=10.0  +MOVJ EC00324
SMOVL C00325 BC00325 V=10.0  +MOVJ EC00325
SMOVL C00326 BC00326 V=10.0  +MOVJ EC00326
SMOVL C00327 BC00327 V=10.0  +MOVJ EC00327
SMOVL C00328 BC00328 V=10.0  +MOVJ EC00328
ARCOF
SMOVL C00329 BC00329 V=400.0  +MOVJ EC00329
SMOVL C00330 BC00330 V=400.0  +MOVJ EC00330
SMOVL C00331 BC00331 V=1000.0  +MOVJ EC00331
SFTOF3D
'Path W948
SFTOF3D
SFTON3D P033
SMOVL C00332 BC00332 V=166.7 PL=0  +MOVJ EC00332
SREFP 1 C00333 BC00333  +REFP EC00333
SREFP 2 C00334 BC00334  +REFP EC00334
ARCON
SMOVL C00335 BC00335 V=10.0  +MOVJ EC00335
ARCOF
SMOVL C00336 BC00336 V=400.0  +MOVJ EC00336
SMOVL C00337 BC00337 V=400.0  +MOVJ EC00337
SMOVL C00338 BC00338 V=1000.0  +MOVJ EC00338
SFTOF3D
'12
'Path W945
SFTOF3D
SFTON3D P034
MOVJ C00339 BC00339 VJ=100.00  +MOVJ EC00339 VJ=100.00
SMOVL C00340 BC00340 V=400.0  +MOVJ EC00340
SMOVL C00341 BC00341 V=166.7 PL=0  +MOVJ EC00341
SREFP 1 C00342 BC00342  +REFP EC00342
SREFP 2 C00343 BC00343  +REFP EC00343
MACRO1 MJ#(0) ARGF14
ARCON
COMM SWVON WEV#(23)
SMOVL C00344 BC00344 V=9.2  +MOVJ EC00344
ARCOF
SWVOF
SMOVL C00345 BC00345 V=400.0  +MOVJ EC00345
SMOVL C00346 BC00346 V=1000.0  +MOVJ EC00346
SFTOF3D
'Path W949
SFTOF3D
SFTON3D P036
MOVJ C00347 BC00347 VJ=100.00  +MOVJ EC00347 VJ=100.00
SMOVL C00348 BC00348 V=166.7 PL=0  +MOVJ EC00348
SREFP 1 C00349 BC00349  +REFP EC00349
SREFP 2 C00350 BC00350  +REFP EC00350
MACRO1 MJ#(0) ARGF14
ARCON
SMOVL C00351 BC00351 V=10.0  +MOVJ EC00351
SMOVL C00352 BC00352 V=10.0  +MOVJ EC00352
SMOVL C00353 BC00353 V=10.0  +MOVJ EC00353
SMOVL C00354 BC00354 V=10.0  +MOVJ EC00354
ARCOF
SMOVL C00355 BC00355 V=400.0  +MOVJ EC00355
SMOVL C00356 BC00356 V=1000.0  +MOVJ EC00356
SFTOF3D
'Path W950
SFTOF3D
SFTON3D P036
MOVJ C00357 BC00357 VJ=100.00  +MOVJ EC00357 VJ=100.00
SMOVL C00358 BC00358 V=1000.0  +MOVJ EC00358
SFTOF3D
MOVJ C00359 BC00359 VJ=100.00  +MOVJ EC00359 VJ=10.00
MOVJ C00360 BC00360 VJ=100.00  +MOVJ EC00360 VJ=100.00
'Path W951
SFTOF3D
SFTON3D P036
MOVJ C00361 BC00361 VJ=100.00  +MOVJ EC00361 VJ=100.00
SMOVL C00362 BC00362 V=400.0  +MOVJ EC00362
SMOVL C00363 BC00363 V=166.7 PL=0  +MOVJ EC00363
SREFP 1 C00364 BC00364  +REFP EC00364
SREFP 2 C00365 BC00365  +REFP EC00365
MACRO1 MJ#(0) ARGF9
ARCON
SMOVL C00366 BC00366 V=10.0  +MOVJ EC00366
ARCOF
SMOVL C00367 BC00367 V=400.0  +MOVJ EC00367
SMOVL C00368 BC00368 V=1000.0  +MOVJ EC00368
SFTOF3D
MOVJ C00369 BC00369 VJ=100.00  +MOVJ EC00369 VJ=100.00
MOVJ C00370 BC00370 VJ=100.00  +MOVJ EC00370 VJ=100.00
'13
'Path W952
SFTOF3D
SFTON3D P041
SMOVL C00371 BC00371 V=400.0  +MOVJ EC00371
SMOVL C00372 BC00372 V=166.7  +MOVJ EC00372
ARCON
COMM SWVON WEV#(10)
SMOVL C00373 BC00373 V=6.7  +MOVJ EC00373
SMOVL C00374 BC00374 V=6.7  +MOVJ EC00374
ARCOF
SWVOF
SMOVL C00375 BC00375 V=200.0  +MOVJ EC00375
SFTON3D P041
SMOVL C00376 BC00376 V=166.7 PL=0  +MOVJ EC00376
SREFP 1 C00377 BC00377  +REFP EC00377
SREFP 2 C00378 BC00378  +REFP EC00378
COMM MACRO1 MJ#(0) ARGF14
'speed bylo v=65
MACRO1 MJ#(0) ARGF9
ARCON
COMM SWVON WEV#(10)
COMM SMOVL C00379 BC00379 V=6.7  +MOVJ EC00379
SFTON3D P042
SMOVL C00380 BC00380 V=6.7  +MOVJ EC00380
SFTON3D P062
SMOVL C00381 BC00381 V=6.7  +MOVJ EC00381
SFTON3D P063
SMOVL C00382 BC00382 V=6.7  +MOVJ EC00382
ARCOF
SWVOF
SMOVL C00383 BC00383 V=333.3  +MOVJ EC00383
SMOVL C00384 BC00384 V=400.0  +MOVJ EC00384
SFTOF3D
MOVJ C00385 BC00385 VJ=100.00  +MOVJ EC00385 VJ=10.00
MOVJ C00386 BC00386 VJ=100.00  +MOVJ EC00386 VJ=100.00
SMOVL C00387 BC00387 V=1000.0  +MOVJ EC00387
SFTON3D P055
MACRO1 MJ#(0) ARGF9
SMOVL C00388 BC00388 V=333.3  +MOVJ EC00388
ARCON
SMOVL C00389 BC00389 V=11.7  +MOVJ EC00389
ARCOF
SFTOF3D
SMOVL C00390 BC00390 V=333.3  +MOVJ EC00390
MOVJ C00391 BC00391 VJ=100.00  +MOVJ EC00391 VJ=20.00
MOVJ C00392 BC00392 VJ=100.00  +MOVJ EC00392 VJ=20.00
SFTON3D P060
SMOVL C00393 BC00393 V=166.7  +MOVJ EC00393
ARCON
SMOVL C00394 BC00394 V=11.7  +MOVJ EC00394
SMOVL C00395 BC00395 V=11.7  +MOVJ EC00395
ARCOF
SMOVL C00396 BC00396 V=333.3  +MOVJ EC00396
SFTOF3D
MOVJ C00397 BC00397 VJ=100.00  +MOVJ EC00397 VJ=10.00
MOVJ C00398 BC00398 VJ=100.00  +MOVJ EC00398 VJ=10.00
'Path W954
SFTOF3D
SFTON3D P037
MOVJ C00399 BC00399 VJ=100.00  +MOVJ EC00399 VJ=100.00
SMOVL C00400 BC00400 V=400.0  +MOVJ EC00400
SMOVL C00401 BC00401 V=166.7 PL=0  +MOVJ EC00401
SREFP 1 C00402 BC00402  +REFP EC00402
SREFP 2 C00403 BC00403  +REFP EC00403
MACRO1 MJ#(0) ARGF14
COMM ARCON
SMOVL C00404 BC00404 V=10.0  +MOVJ EC00404
SMOVL C00405 BC00405 V=10.0  +MOVJ EC00405
ARCOF
SMOVL C00406 BC00406 V=400.0  +MOVJ EC00406
SMOVL C00407 BC00407 V=1000.0  +MOVJ EC00407
SFTOF3D
'Path W955
SFTOF3D
SFTON3D P037
SMOVL C00408 BC00408 V=400.0  +MOVJ EC00408
SMOVL C00409 BC00409 V=133.3 PL=0  +MOVJ EC00409
SREFP 1 C00410 BC00410  +REFP EC00410
SREFP 2 C00411 BC00411  +REFP EC00411
MACRO1 MJ#(0) ARGF14
COMM ARCON
SMOVL C00412 BC00412 V=10.0  +MOVJ EC00412
ARCOF
SMOVL C00413 BC00413 V=400.0  +MOVJ EC00413
SFTOF3D
MOVJ C00414 BC00414 VJ=100.00  +MOVJ EC00414 VJ=100.00
MOVJ C00415 BC00415 VJ=100.00  +MOVJ EC00415 VJ=50.00
'Path W956
SFTOF3D
SFTON3D P037
MOVJ C00416 BC00416 VJ=100.00  +MOVJ EC00416 VJ=100.00
SMOVL C00417 BC00417 V=400.0  +MOVJ EC00417
SMOVL C00418 BC00418 V=133.3 PL=0  +MOVJ EC00418
SREFP 1 C00419 BC00419  +REFP EC00419
SREFP 2 C00420 BC00420  +REFP EC00420
MACRO1 MJ#(0) ARGF14
COMM ARCON
SMOVL C00421 BC00421 V=10.0  +MOVJ EC00421
ARCOF
SMOVL C00422 BC00422 V=400.0  +MOVJ EC00422
SMOVL C00423 BC00423 V=1000.0  +MOVJ EC00423
SFTOF3D
'17
MOVJ C00424 BC00424 VJ=100.00  +MOVJ EC00424 VJ=100.00
MOVJ C00425 BC00425 VJ=100.00  +MOVJ EC00425 VJ=100.00
'Path W957
SFTOF3D
SFTON3D P040
SMOVL C00426 BC00426 V=166.7 PL=0  +MOVJ EC00426
SREFP 1 C00427 BC00427  +REFP EC00427
SREFP 2 C00428 BC00428  +REFP EC00428
MACRO1 MJ#(0) ARGF14
ARCON
SMOVL C00429 BC00429 V=10.0  +MOVJ EC00429
ARCOF
SMOVL C00430 BC00430 V=400.0  +MOVJ EC00430
SMOVL C00431 BC00431 V=333.3  +MOVJ EC00431
SFTOF3D
'Path W958
SFTOF3D
SFTON3D P040
SMOVL C00432 BC00432 V=166.7 PL=0  +MOVJ EC00432
SREFP 1 C00433 BC00433  +REFP EC00433
SREFP 2 C00434 BC00434  +REFP EC00434
MACRO1 MJ#(0) ARGF14
ARCON
SMOVL C00435 BC00435 V=10.0  +MOVJ EC00435
ARCOF
SMOVL C00436 BC00436 V=400.0  +MOVJ EC00436
SFTOF3D
MOVJ C00437 BC00437 VJ=100.00  +MOVJ EC00437 VJ=100.00
'Path W959
SFTOF3D
SFTON3D P040
COMM MOVJ C00438 BC00438 VJ=100.00  +MOVJ EC00438 VJ=100.00
COMM SMOVL C00439 BC00439 V=400.0  +MOVJ EC00439
COMM SMOVL C00440 BC00440 V=100.0 PL=0  +MOVJ EC00440
COMM SREFP 1 C00441 BC00441  +REFP EC00441
COMM SREFP 2 C00442 BC00442  +REFP EC00442
COMM MACRO1 MJ#(0) ARGF0
COMM ARCON
COMM SMOVL C00443 BC00443 V=10.0  +MOVJ EC00443
COMM SMOVL C00444 BC00444 V=10.0  +MOVJ EC00444
COMM SMOVL C00445 BC00445 V=10.0  +MOVJ EC00445
COMM ARCOF
COMM SMOVL C00446 BC00446 V=400.0  +MOVJ EC00446
COMM SMOVL C00447 BC00447 V=1000.0  +MOVJ EC00447
SFTOF3D
'18
'Path W960
SFTOF3D
MOVJ C00448 BC00448 VJ=100.00  +MOVJ EC00448 VJ=100.00
MOVJ C00449 BC00449 VJ=100.00  +MOVJ EC00449 VJ=15.00
MOVJ C00450 BC00450 VJ=100.00  +MOVJ EC00450 VJ=15.00
SMOVL C00451 BC00451 V=400.0  +MOVJ EC00451
SFTON3D P050
SMOVL C00452 BC00452 V=166.7 PL=0  +MOVJ EC00452
SREFP 1 C00453 BC00453  +REFP EC00453
SREFP 2 C00454 BC00454  +REFP EC00454
MACRO1 MJ#(0) ARGF14
COMM ARCON
SMOVL C00455 BC00455 V=9.2  +MOVJ EC00455
SMOVL C00456 BC00456 V=9.2  +MOVJ EC00456
SMOVL C00457 BC00457 V=9.2  +MOVJ EC00457
SMOVL C00458 BC00458 V=9.2  +MOVJ EC00458
SMOVL C00459 BC00459 V=9.2  +MOVJ EC00459
ARCOF
SMOVL C00460 BC00460 V=400.0  +MOVJ EC00460
SMOVL C00461 BC00461 V=1000.0  +MOVJ EC00461
SFTOF3D
'19
MOVJ C00462 BC00462 VJ=100.00  +MOVJ EC00462 VJ=10.00
MOVJ C00463 BC00463 VJ=100.00  +MOVJ EC00463 VJ=100.00
'Path W962
SFTOF3D
SFTON3D P035
MOVJ C00464 BC00464 VJ=100.00  +MOVJ EC00464 VJ=100.00
SMOVL C00465 BC00465 V=400.0  +MOVJ EC00465
SMOVL C00466 BC00466 V=166.7 PL=0  +MOVJ EC00466
SREFP 1 C00467 BC00467  +REFP EC00467
SREFP 2 C00468 BC00468  +REFP EC00468
ARCON
COMM SWVON WEV#(21)
SMOVL C00469 BC00469 V=9.2  +MOVJ EC00469
ARCOF
SWVOF
SMOVL C00470 BC00470 V=400.0  +MOVJ EC00470
SMOVL C00471 BC00471 V=1000.0  +MOVJ EC00471
SFTOF3D
'20
MOVJ C00472 BC00472 VJ=100.00  +MOVJ EC00472 VJ=100.00
MOVJ C00473 BC00473 VJ=100.00  +MOVJ EC00473 VJ=10.00
MOVJ C00474 BC00474 VJ=100.00  +MOVJ EC00474 VJ=100.00
'Path W963
SFTOF3D
SFTON3D P052
SMOVL C00475 BC00475 V=400.0  +MOVJ EC00475
SMOVL C00476 BC00476 V=166.7 PL=0  +MOVJ EC00476
SREFP 1 C00477 BC00477  +REFP EC00477
SREFP 2 C00478 BC00478  +REFP EC00478
MACRO1 MJ#(0) ARGF6
ARCON
SMOVL C00479 BC00479 V=7.5  +MOVJ EC00479
SMOVL C00480 BC00480 V=7.5  +MOVJ EC00480
SMOVL C00481 BC00481 V=7.5  +MOVJ EC00481
ARCOF
SMOVL C00482 BC00482 V=400.0  +MOVJ EC00482
SFTOF3D
'Path W964
SFTOF3D
SFTON3D P052
SMOVL C00483 BC00483 V=500.0  +MOVJ EC00483
SFTOF3D
SFTON3D P052
SMOVL C00484 BC00484 V=500.0  +MOVJ EC00484
SMOVL C00485 BC00485 V=166.7 PL=0  +MOVJ EC00485
SREFP 1 C00486 BC00486  +REFP EC00486
SREFP 2 C00487 BC00487  +REFP EC00487
MACRO1 MJ#(0) ARGF6
ARCON
SMOVL C00488 BC00488 V=9.2  +MOVJ EC00488
ARCOF
SMOVL C00489 BC00489 V=400.0  +MOVJ EC00489
SMOVL C00490 BC00490 V=1000.0  +MOVJ EC00490
SFTOF3D
'Path W967
SFTOF3D
SFTON3D P052
MOVJ C00491 BC00491 VJ=100.00  +MOVJ EC00491 VJ=10.00
MOVJ C00492 BC00492 VJ=100.00  +MOVJ EC00492 VJ=100.00
SMOVL C00493 BC00493 V=500.0  +MOVJ EC00493
SMOVL C00494 BC00494 V=166.7 PL=0  +MOVJ EC00494
SREFP 1 C00495 BC00495  +REFP EC00495
SREFP 2 C00496 BC00496  +REFP EC00496
MACRO1 MJ#(0) ARGF6
ARCON
SMOVL C00497 BC00497 V=10.0  +MOVJ EC00497
ARCOF
SMOVL C00498 BC00498 V=500.0  +MOVJ EC00498
SFTOF3D
MOVJ C00499 BC00499 VJ=100.00  +MOVJ EC00499 VJ=100.00
'21
MOVJ C00500 BC00500 VJ=100.00  +MOVJ EC00500 VJ=100.00
MOVJ C00501 BC00501 VJ=100.00  +MOVJ EC00501 VJ=100.00
'Path W968
SFTOF3D
SFTON3D P061
SMOVL C00502 BC00502 V=500.0  +MOVJ EC00502
SREFP 1 C00503 BC00503  +REFP EC00503
SREFP 2 C00504 BC00504  +REFP EC00504
SMOVL C00505 BC00505 V=166.7 PL=0  +MOVJ EC00505
MACRO1 MJ#(0) ARGF9
ARCON
SFTON3D P064
SMOVL C00506 BC00506 V=10.8  +MOVJ EC00506
SMOVL C00507 BC00507 V=10.8  +MOVJ EC00507
SFTON3D P031
SMOVL C00508 BC00508 V=10.8 PL=0  +MOVJ EC00508
SFTON3D P032
SMOVL C00509 BC00509 V=10.8  +MOVJ EC00509
ARCOF
SMOVL C00510 BC00510 V=400.0  +MOVJ EC00510
SFTOF3D
MOVJ C00511 BC00511 VJ=100.00  +MOVJ EC00511 VJ=100.00
MOVJ C00512 BC00512 VJ=100.00  +MOVJ EC00512 VJ=100.00
MOVJ C00513 BC00513 VJ=100.00  +MOVJ EC00513 VJ=100.00
CALL JOB:CLEAN-R1_KM_3P
'cut_wire_dol
'cut_wire_dol
'cut_wire_dol
MOVJ C00514 BC00514 VJ=100.00  +MOVJ EC00514 VJ=100.00
'Path S1328
SFTOF3D
MOVJ C00515 BC00515 VJ=100.00  +MOVJ EC00515 VJ=100.00
MOVJ C00516 BC00516 VJ=100.00  +MOVJ EC00516 VJ=100.00
MOVJ C00517 BC00517 VJ=15.00  +MOVJ EC00517 VJ=100.00
MOVL C00518 BC00518 V=333.3  +MOVJ EC00518 VJ=100.00
SFTOF3D
SMOVL C00519 BC00519 V=166.7  +MOVJ EC00519
SREFP 3 C00520 BC00520  +REFP EC00520
CALL JOB:SEARCH-R1-S13D
SET P023 P006
SFTON3D P023
SMOVL C00521 BC00521 V=166.7  +MOVJ EC00521
SMOVL C00522 BC00522 V=166.7  +MOVJ EC00522
SMOVL C00523 BC00523 V=166.7  +MOVJ EC00523
SREFP 3 C00524 BC00524  +REFP EC00524
CALL JOB:SEARCH-R1-S13D
SET P023 P006
SFTON3D P023
SMOVL C00525 BC00525 V=166.7  +MOVJ EC00525
MOVL C00526 BC00526 V=400.0  +MOVJ EC00526 VJ=100.00
MOVJ C00527 BC00527 VJ=100.00  +MOVJ EC00527 VJ=100.00
MOVJ C00528 BC00528 VJ=100.00  +MOVJ EC00528 VJ=100.00
'Path S1331
SFTOF3D
MOVL C00529 BC00529 V=166.7  +MOVJ EC00529 VJ=100.00
SMOVL C00530 BC00530 V=166.7  +MOVJ EC00530
SREFP 3 C00531 BC00531  +REFP EC00531
CALL JOB:SEARCH-R1-S13D
SET P022 P006
SFTON3D P022
SMOVL C00532 BC00532 V=166.7  +MOVJ EC00532
SMOVL C00533 BC00533 V=166.7  +MOVJ EC00533
